LIN {X 0,Y 524.033,Z 442.422,A -85,B 0,C 180,E1 -4780.038,E2 -4780.038} C_VEL
LIN {X 0,Y 524.328,Z 431.907,A -85,B 0,C 180,E1 -4781.009,E2 -4781.009} C_VEL
LIN {X 0,Y 524.611,Z 421.558,A -85,B 0,C 180,E1 -4781.783,E2 -4781.783} C_VEL
LIN {X 0,Y 524.883,Z 410.111,A -85,B 0,C 180,E1 -4782.466,E2 -4782.466} C_VEL
LIN {X 0,Y 525.105,Z 398.418,A -85,B 0,C 180,E1 -4783.001,E2 -4783.001} C_VEL
LIN {X 0,Y 525.367,Z 384.955,A -85,B 0,C 180,E1 -4783.438,E2 -4783.438} C_VEL
LIN {X 0,Y 525.555,Z 371.649,A -85,B 0,C 180,E1 -4783.704,E2 -4783.704} C_VEL
LIN {X 0,Y 525.723,Z 278.906,A -85,B 0,C 180,E1 -4784.981,E2 -4784.981} C_VEL
LIN {X 0,Y 524.283,Z 268.974,A -85,B 0,C 180,E1 -4785.168,E2 -4785.168} C_VEL
LIN {X 0,Y 524.683,Z 247.787,A -85,B 0,C 180,E1 -4788.304,E2 -4788.304} C_VEL
LIN {X 0,Y 525.117,Z 227.261,A -85,B 0,C 180,E1 -4791.386,E2 -4791.386} C_VEL
LIN {X 0,Y 525.445,Z 212.359,A -85,B 0,C 180,E1 -4793.653,E2 -4793.653} C_VEL
LIN {X 0,Y 523.986,Z 204.215,A -85,B 0,C 180,E1 -4794.988,E2 -4794.988} C_VEL
LIN {X 0,Y 523.957,Z 204.223,A -85,B 0,C 180,E1 -4797.995,E2 -4797.995} C_VEL
LIN {X 0,Y 523.928,Z 204.217,A -85,B 0,C 180,E1 -4800.851,E2 -4800.851} C_VEL
LIN {X 0,Y 523.944,Z 204.22,A -85,B 0,C 180,E1 -4803.731,E2 -4803.731} C_VEL
LIN {X 0,Y 523.901,Z 204.224,A -85,B 0,C 180,E1 -4806.4,E2 -4806.4} C_VEL
LIN {X 0,Y 523.899,Z 204.221,A -85,B 0,C 180,E1 -4809.081,E2 -4809.081} C_VEL
LIN {X 0,Y 523.929,Z 204.223,A -85,B 0,C 180,E1 -4812.115,E2 -4812.115} C_VEL
LIN {X 0,Y 523.925,Z 204.219,A -85,B 0,C 180,E1 -4815.305,E2 -4815.305} C_VEL
LIN {X 0,Y 523.949,Z 204.214,A -85,B 0,C 180,E1 -4818.683,E2 -4818.683} C_VEL
LIN {X 0,Y 523.919,Z 204.219,A -85,B 0,C 180,E1 -4821.072,E2 -4821.072} C_VEL
LIN {X 0,Y 523.891,Z 204.229,A -85,B 0,C 180,E1 -4823.824,E2 -4823.824} C_VEL
LIN {X 0,Y 523.902,Z 204.22,A -85,B 0,C 180,E1 -4826.632,E2 -4826.632} C_VEL
LIN {X 0,Y 523.92,Z 204.223,A -85,B 0,C 180,E1 -4829.353,E2 -4829.353} C_VEL
LIN {X 0,Y 523.936,Z 204.217,A -85,B 0,C 180,E1 -4832.277,E2 -4832.277} C_VEL
LIN {X 0,Y 523.908,Z 204.22,A -85,B 0,C 180,E1 -4834.579,E2 -4834.579} C_VEL
LIN {X 0,Y 523.911,Z 204.223,A -85,B 0,C 180,E1 -4837.106,E2 -4837.106} C_VEL
LIN {X 0,Y 523.928,Z 204.22,A -85,B 0,C 180,E1 -4839.863,E2 -4839.863} C_VEL
LIN {X 0,Y 523.945,Z 204.217,A -85,B 0,C 180,E1 -4842.836,E2 -4842.836} C_VEL
LIN {X 0,Y 523.95,Z 204.222,A -85,B 0,C 180,E1 -4845.235,E2 -4845.235} C_VEL
LIN {X 0,Y 523.963,Z 204.213,A -85,B 0,C 180,E1 -4848.393,E2 -4848.393} C_VEL
LIN {X 0,Y 523.954,Z 204.219,A -85,B 0,C 180,E1 -4851.515,E2 -4851.515} C_VEL
LIN {X 0,Y 523.997,Z 204.21,A -85,B 0,C 180,E1 -4853.84,E2 -4853.84} C_VEL
LIN {X 0,Y 524.024,Z 204.211,A -85,B 0,C 180,E1 -4856.925,E2 -4856.925} C_VEL
LIN {X 0,Y 524.051,Z 204.202,A -85,B 0,C 180,E1 -4860,E2 -4860} C_VEL
LIN {X 0,Y 524.022,Z 204.214,A -85,B 0,C 180,E1 -4863.075,E2 -4863.075} C_VEL
LIN {X 0,Y 523.98,Z 204.211,A -85,B 0,C 180,E1 -4866.16,E2 -4866.16} C_VEL
LIN {X 0,Y 523.95,Z 204.218,A -85,B 0,C 180,E1 -4869.262,E2 -4869.262} C_VEL
LIN {X 0,Y 523.968,Z 204.212,A -85,B 0,C 180,E1 -4871.752,E2 -4871.752} C_VEL
LIN {X 0,Y 523.936,Z 204.222,A -85,B 0,C 180,E1 -4875.053,E2 -4875.053} C_VEL
LIN {X 0,Y 523.917,Z 204.219,A -85,B 0,C 180,E1 -4877.97,E2 -4877.97} C_VEL
LIN {X 0,Y 523.92,Z 204.222,A -85,B 0,C 180,E1 -4880.412,E2 -4880.412} C_VEL
LIN {X 0,Y 523.892,Z 204.227,A -85,B 0,C 180,E1 -4882.894,E2 -4882.894} C_VEL
LIN {X 0,Y 523.936,Z 204.217,A -85,B 0,C 180,E1 -4886.022,E2 -4886.022} C_VEL
LIN {X 0,Y 523.895,Z 204.226,A -85,B 0,C 180,E1 -4888.877,E2 -4888.877} C_VEL
LIN {X 0,Y 523.885,Z 204.222,A -85,B 0,C 180,E1 -4891.546,E2 -4891.546} C_VEL
LIN {X 0,Y 523.9,Z 204.227,A -85,B 0,C 180,E1 -4894.292,E2 -4894.292} C_VEL
LIN {X 0,Y 523.871,Z 204.225,A -85,B 0,C 180,E1 -4897.135,E2 -4897.135} C_VEL
LIN {X 0,Y 523.899,Z 204.226,A -85,B 0,C 180,E1 -4900.133,E2 -4900.133} C_VEL
LIN {X 0,Y 523.901,Z 204.228,A -85,B 0,C 180,E1 -4902.462,E2 -4902.462} C_VEL
LIN {X 0,Y 523.91,Z 204.219,A -85,B 0,C 180,E1 -4905.314,E2 -4905.314} C_VEL
LIN {X 0,Y 523.884,Z 204.223,A -85,B 0,C 180,E1 -4906.944,E2 -4906.944} C_VEL
LIN {X 0,Y 523.222,Z 204.306,A -85,B 0,C 180,E1 -4907.585,E2 -4907.585} C_VEL
LIN {X 0,Y 520.38,Z 204.669,A -85,B 0,C 180,E1 -4908.627,E2 -4908.627} C_VEL
LIN {X 0,Y 517.974,Z 204.973,A -85,B 0,C 180,E1 -4909.466,E2 -4909.466} C_VEL
LIN {X 0,Y 516.938,Z 205.098,A -85,B 0,C 180,E1 -4910.114,E2 -4910.114} C_VEL
LIN {X 0,Y 516.852,Z 205.106,A -85,B 0,C 180,E1 -4910.334,E2 -4910.334} C_VEL
LIN {X 0,Y 516.859,Z 205.098,A -85,B 0,C 180,E1 -4913.345,E2 -4913.345} C_VEL
LIN {X 0,Y 516.888,Z 205.103,A -85,B 0,C 180,E1 -4916.124,E2 -4916.124} C_VEL
LIN {X 0,Y 516.871,Z 205.096,A -85,B 0,C 180,E1 -4918.939,E2 -4918.939} C_VEL
LIN {X 0,Y 516.897,Z 205.096,A -85,B 0,C 180,E1 -4921.588,E2 -4921.588} C_VEL
LIN {X 0,Y 516.914,Z 205.096,A -85,B 0,C 180,E1 -4924.214,E2 -4924.214} C_VEL
LIN {X 0,Y 516.846,Z 205.099,A -85,B 0,C 180,E1 -4926.779,E2 -4926.779} C_VEL
LIN {X 0,Y 516.926,Z 205.096,A -85,B 0,C 180,E1 -4929.735,E2 -4929.735} C_VEL
LIN {X 0,Y 516.884,Z 205.095,A -85,B 0,C 180,E1 -4932.598,E2 -4932.598} C_VEL
LIN {X 0,Y 516.928,Z 205.09,A -85,B 0,C 180,E1 -4935.032,E2 -4935.032} C_VEL
LIN {X 0,Y 516.961,Z 205.087,A -85,B 0,C 180,E1 -4938.236,E2 -4938.236} C_VEL
LIN {X 0,Y 516.959,Z 205.09,A -85,B 0,C 180,E1 -4941.402,E2 -4941.402} C_VEL
LIN {X 0,Y 517.019,Z 205.081,A -85,B 0,C 180,E1 -4944.542,E2 -4944.542} C_VEL
LIN {X 0,Y 516.866,Z 205.164,A -85,B 0,C 180,E1 -4946.006,E2 -4946.006} C_VEL
LIN {X 0,Y 517.422,Z 209.6,A -85,B 0,C 180,E1 -4946.887,E2 -4946.887} C_VEL
LIN {X 0,Y 517.24,Z 224.307,A -85,B 0,C 180,E1 -4949.697,E2 -4949.697} C_VEL
LIN {X 0,Y 519.169,Z 234.742,A -85,B 0,C 180,E1 -4949.904,E2 -4949.904} C_VEL
LIN {X 0,Y 518.648,Z 331.01,A -85,B 0,C 180,E1 -4951.263,E2 -4951.263} C_VEL
LIN {X 0,Y 518.467,Z 343.297,A -85,B 0,C 180,E1 -4951.579,E2 -4951.579} C_VEL
LIN {X 0,Y 518.269,Z 356.555,A -85,B 0,C 180,E1 -4952.09,E2 -4952.09} C_VEL
LIN {X 0,Y 517.968,Z 368.557,A -85,B 0,C 180,E1 -4952.723,E2 -4952.723} C_VEL
LIN {X 0,Y 517.629,Z 379.969,A -85,B 0,C 180,E1 -4953.504,E2 -4953.504} C_VEL
LIN {X 0,Y 517.351,Z 390.246,A -85,B 0,C 180,E1 -4954.383,E2 -4954.383} C_VEL
LIN {X 0,Y 517.064,Z 398.689,A -85,B 0,C 180,E1 -4955.265,E2 -4955.265} C_VEL
LIN {X 0,Y 516.856,Z 406.477,A -85,B 0,C 180,E1 -4956.246,E2 -4956.246} C_VEL
LIN {X 0,Y 516.683,Z 414.099,A -85,B 0,C 180,E1 -4957.425,E2 -4957.425} C_VEL
LIN {X 0,Y 516.521,Z 420.242,A -85,B 0,C 180,E1 -4958.608,E2 -4958.608} C_VEL
LIN {X 0,Y 516.42,Z 425.127,A -85,B 0,C 180,E1 -4959.795,E2 -4959.795} C_VEL
LIN {X 0,Y 516.338,Z 428.896,A -85,B 0,C 180,E1 -4960.986,E2 -4960.986} C_VEL
LIN {X 0,Y 516.291,Z 430.844,A -85,B 0,C 180,E1 -4961.782,E2 -4961.782} C_VEL
LIN {X 0,Y 516.23,Z 432.359,A -85,B 0,C 180,E1 -4962.582,E2 -4962.582} C_VEL
LIN {X 0,Y 516.205,Z 433.411,A -85,B 0,C 180,E1 -4963.383,E2 -4963.383} C_VEL
LIN {X 0,Y 516.249,Z 434.294,A -85,B 0,C 180,E1 -4964.859,E2 -4964.859} C_VEL
LIN {X 0,Y 516.174,Z 434.133,A -85,B 0,C 180,E1 -4965.802,E2 -4965.802} C_VEL
LIN {X 0,Y 516.195,Z 433.514,A -85,B 0,C 180,E1 -4966.613,E2 -4966.613} C_VEL
LIN {X 0,Y 516.247,Z 432.135,A -85,B 0,C 180,E1 -4967.645,E2 -4967.645} C_VEL
LIN {X 0,Y 516.303,Z 429.017,A -85,B 0,C 180,E1 -4969.068,E2 -4969.068} C_VEL
LIN {X 0,Y 516.402,Z 424.901,A -85,B 0,C 180,E1 -4970.367,E2 -4970.367} C_VEL
LIN {X 0,Y 516.481,Z 419.948,A -85,B 0,C 180,E1 -4971.555,E2 -4971.555} C_VEL
LIN {X 0,Y 516.685,Z 413.32,A -85,B 0,C 180,E1 -4972.808,E2 -4972.808} C_VEL
LIN {X 0,Y 516.912,Z 404.823,A -85,B 0,C 180,E1 -4974.071,E2 -4974.071} C_VEL
LIN {X 0,Y 517.164,Z 396.005,A -85,B 0,C 180,E1 -4975.129,E2 -4975.129} C_VEL
LIN {X 0,Y 517.466,Z 386.153,A -85,B 0,C 180,E1 -4976.087,E2 -4976.087} C_VEL
LIN {X 0,Y 517.771,Z 375.246,A -85,B 0,C 180,E1 -4976.936,E2 -4976.936} C_VEL
LIN {X 0,Y 518.116,Z 363.348,A -85,B 0,C 180,E1 -4977.668,E2 -4977.668} C_VEL
LIN {X 0,Y 518.317,Z 352.206,A -85,B 0,C 180,E1 -4978.195,E2 -4978.195} C_VEL
LIN {X 0,Y 518.52,Z 339.67,A -85,B 0,C 180,E1 -4978.622,E2 -4978.622} C_VEL
LIN {X 0,Y 518.636,Z 326.636,A -85,B 0,C 180,E1 -4978.905,E2 -4978.905} C_VEL
LIN {X 0,Y 519.051,Z 233.834,A -85,B 0,C 180,E1 -4980.204,E2 -4980.204} C_VEL
LIN {X 0,Y 517.237,Z 224.156,A -85,B 0,C 180,E1 -4980.397,E2 -4980.397} C_VEL
LIN {X 0,Y 517.378,Z 209.592,A -85,B 0,C 180,E1 -4983.143,E2 -4983.143} C_VEL
LIN {X 0,Y 516.965,Z 205.092,A -85,B 0,C 180,E1 -4984.019,E2 -4984.019} C_VEL
LIN {X 0,Y 516.873,Z 205.103,A -85,B 0,C 180,E1 -4986.744,E2 -4986.744} C_VEL
LIN {X 0,Y 516.891,Z 205.098,A -85,B 0,C 180,E1 -4989.718,E2 -4989.718} C_VEL
LIN {X 0,Y 516.894,Z 205.099,A -85,B 0,C 180,E1 -4992.759,E2 -4992.759} C_VEL
LIN {X 0,Y 516.907,Z 205.094,A -85,B 0,C 180,E1 -4995.009,E2 -4995.009} C_VEL
LIN {X 0,Y 516.905,Z 205.099,A -85,B 0,C 180,E1 -4998.396,E2 -4998.396} C_VEL
LIN {X 0,Y 516.866,Z 205.098,A -85,B 0,C 180,E1 -5001.283,E2 -5001.283} C_VEL
LIN {X 0,Y 516.869,Z 205.102,A -85,B 0,C 180,E1 -5004.22,E2 -5004.22} C_VEL
LIN {X 0,Y 516.875,Z 205.096,A -85,B 0,C 180,E1 -5007.052,E2 -5007.052} C_VEL
LIN {X 0,Y 516.877,Z 205.102,A -85,B 0,C 180,E1 -5009.796,E2 -5009.796} C_VEL
LIN {X 0,Y 516.904,Z 205.093,A -85,B 0,C 180,E1 -5012.466,E2 -5012.466} C_VEL
LIN {X 0,Y 516.893,Z 205.092,A -85,B 0,C 180,E1 -5015.071,E2 -5015.071} C_VEL
LIN {X 0,Y 516.884,Z 205.102,A -85,B 0,C 180,E1 -5017.622,E2 -5017.622} C_VEL
LIN {X 0,Y 516.902,Z 205.095,A -85,B 0,C 180,E1 -5020.129,E2 -5020.129} C_VEL
LIN {X 0,Y 516.912,Z 205.089,A -85,B 0,C 180,E1 -5022.596,E2 -5022.596} C_VEL
LIN {X 0,Y 516.918,Z 205.093,A -85,B 0,C 180,E1 -5025.03,E2 -5025.03} C_VEL
LIN {X 0,Y 516.933,Z 205.089,A -85,B 0,C 180,E1 -5028.233,E2 -5028.233} C_VEL
LIN {X 0,Y 516.94,Z 205.093,A -85,B 0,C 180,E1 -5031.399,E2 -5031.399} C_VEL
LIN {X 0,Y 516.985,Z 205.085,A -85,B 0,C 180,E1 -5033.757,E2 -5033.757} C_VEL
LIN {X 0,Y 516.984,Z 205.082,A -85,B 0,C 180,E1 -5036.883,E2 -5036.883} C_VEL
LIN {X 0,Y 517.044,Z 205.073,A -85,B 0,C 180,E1 -5040,E2 -5040} C_VEL
LIN {X 0,Y 516.982,Z 205.088,A -85,B 0,C 180,E1 -5043.117,E2 -5043.117} C_VEL
LIN {X 0,Y 516.967,Z 205.081,A -85,B 0,C 180,E1 -5046.244,E2 -5046.244} C_VEL
LIN {X 0,Y 516.921,Z 205.09,A -85,B 0,C 180,E1 -5049.39,E2 -5049.39} C_VEL
LIN {X 0,Y 516.952,Z 205.085,A -85,B 0,C 180,E1 -5051.825,E2 -5051.825} C_VEL
LIN {X 0,Y 516.912,Z 205.096,A -85,B 0,C 180,E1 -5055.147,E2 -5055.147} C_VEL
LIN {X 0,Y 516.885,Z 205.095,A -85,B 0,C 180,E1 -5058.224,E2 -5058.224} C_VEL
LIN {X 0,Y 516.883,Z 205.101,A -85,B 0,C 180,E1 -5060.703,E2 -5060.703} C_VEL
LIN {X 0,Y 516.855,Z 205.098,A -85,B 0,C 180,E1 -5064.075,E2 -5064.075} C_VEL
LIN {X 0,Y 516.866,Z 205.104,A -85,B 0,C 180,E1 -5066.661,E2 -5066.661} C_VEL
LIN {X 0,Y 516.883,Z 205.095,A -85,B 0,C 180,E1 -5069.525,E2 -5069.525} C_VEL
LIN {X 0,Y 516.871,Z 205.105,A -85,B 0,C 180,E1 -5072.545,E2 -5072.545} C_VEL
LIN {X 0,Y 516.841,Z 205.101,A -85,B 0,C 180,E1 -5075.331,E2 -5075.331} C_VEL
LIN {X 0,Y 516.857,Z 205.1,A -85,B 0,C 180,E1 -5077.944,E2 -5077.944} C_VEL
LIN {X 0,Y 516.867,Z 205.097,A -85,B 0,C 180,E1 -5080.744,E2 -5080.744} C_VEL
LIN {X 0,Y 516.867,Z 205.099,A -85,B 0,C 180,E1 -5082.833,E2 -5082.833} C_VEL
LIN {X 0,Y 516.882,Z 205.096,A -85,B 0,C 180,E1 -5085.009,E2 -5085.009} C_VEL
LIN {X 0,Y 516.89,Z 205.1,A -85,B 0,C 180,E1 -5088.402,E2 -5088.402} C_VEL
LIN {X 0,Y 516.867,Z 205.098,A -85,B 0,C 180,E1 -5091.285,E2 -5091.285} C_VEL
LIN {X 0,Y 516.868,Z 205.105,A -85,B 0,C 180,E1 -5094.222,E2 -5094.222} C_VEL
LIN {X 0,Y 516.889,Z 205.096,A -85,B 0,C 180,E1 -5097.054,E2 -5097.054} C_VEL
LIN {X 0,Y 516.887,Z 205.101,A -85,B 0,C 180,E1 -5099.798,E2 -5099.798} C_VEL
LIN {X 0,Y 516.895,Z 205.099,A -85,B 0,C 180,E1 -5102.467,E2 -5102.467} C_VEL
LIN {X 0,Y 516.93,Z 205.133,A -85,B 0,C 180,E1 -5104.913,E2 -5104.913} C_VEL
LIN {X 0,Y 518.493,Z 214.374,A -85,B 0,C 180,E1 -5106.431,E2 -5106.431} C_VEL
LIN {X 0,Y 517.974,Z 234.682,A -85,B 0,C 180,E1 -5109.539,E2 -5109.539} C_VEL
LIN {X 0,Y 517.563,Z 253.888,A -85,B 0,C 180,E1 -5112.437,E2 -5112.437} C_VEL
LIN {X 0,Y 517.227,Z 268.524,A -85,B 0,C 180,E1 -5114.62,E2 -5114.62} C_VEL
LIN {X 0,Y 519.024,Z 282.03,A -85,B 0,C 180,E1 -5114.87,E2 -5114.87} C_VEL
LIN {X 0,Y 518.593,Z 376.948,A -85,B 0,C 180,E1 -5116.206,E2 -5116.206} C_VEL
LIN {X 0,Y 518.326,Z 390.326,A -85,B 0,C 180,E1 -5116.548,E2 -5116.548} C_VEL
LIN {X 0,Y 518.033,Z 402.555,A -85,B 0,C 180,E1 -5117.015,E2 -5117.015} C_VEL
LIN {X 0,Y 517.801,Z 414.873,A -85,B 0,C 180,E1 -5117.655,E2 -5117.655} C_VEL
LIN {X 0,Y 517.468,Z 426.547,A -85,B 0,C 180,E1 -5118.444,E2 -5118.444} C_VEL
LIN {X 0,Y 517.209,Z 437.038,A -85,B 0,C 180,E1 -5119.33,E2 -5119.33} C_VEL
LIN {X 0,Y 516.917,Z 445.615,A -85,B 0,C 180,E1 -5120.215,E2 -5120.215} C_VEL
LIN {X 0,Y 516.703,Z 453.533,A -85,B 0,C 180,E1 -5121.198,E2 -5121.198} C_VEL
LIN {X 0,Y 516.521,Z 461.27,A -85,B 0,C 180,E1 -5122.376,E2 -5122.376} C_VEL
LIN {X 0,Y 516.389,Z 468.402,A -85,B 0,C 180,E1 -5123.749,E2 -5123.749} C_VEL
LIN {X 0,Y 516.312,Z 473.149,A -85,B 0,C 180,E1 -5124.923,E2 -5124.923} C_VEL
LIN {X 0,Y 516.352,Z 476.781,A -85,B 0,C 180,E1 -5126.097,E2 -5126.097} C_VEL
LIN {X 0,Y 516.283,Z 478.651,A -85,B 0,C 180,E1 -5126.878,E2 -5126.878} C_VEL
LIN {X 0,Y 516.262,Z 480.055,A -85,B 0,C 180,E1 -5127.658,E2 -5127.658} C_VEL
LIN {X 0,Y 516.167,Z 481.667,A -85,B 0,C 180,E1 -5129.219,E2 -5129.219} C_VEL
LIN {X 0,Y 516.167,Z 481.887,A -85,B 0,C 180,E1 -5129.999,E2 -5129.999} C_VEL
LIN {X 0,Y 516.192,Z 481.066,A -85,B 0,C 180,E1 -5131.559,E2 -5131.559} C_VEL
LIN {X 0,Y 516.261,Z 480.072,A -85,B 0,C 180,E1 -5132.339,E2 -5132.339} C_VEL
LIN {X 0,Y 516.282,Z 478.673,A -85,B 0,C 180,E1 -5133.12,E2 -5133.12} C_VEL
LIN {X 0,Y 516.311,Z 475.73,A -85,B 0,C 180,E1 -5134.292,E2 -5134.292} C_VEL
LIN {X 0,Y 516.368,Z 471.744,A -85,B 0,C 180,E1 -5135.465,E2 -5135.465} C_VEL
LIN {X 0,Y 516.387,Z 466.554,A -85,B 0,C 180,E1 -5136.653,E2 -5136.653} C_VEL
LIN {X 0,Y 516.543,Z 460.155,A -85,B 0,C 180,E1 -5137.818,E2 -5137.818} C_VEL
LIN {X 0,Y 516.752,Z 452.102,A -85,B 0,C 180,E1 -5138.996,E2 -5138.996} C_VEL
LIN {X 0,Y 516.948,Z 443.896,A -85,B 0,C 180,E1 -5139.98,E2 -5139.98} C_VEL
LIN {X 0,Y 517.262,Z 433.895,A -85,B 0,C 180,E1 -5140.963,E2 -5140.963} C_VEL
LIN {X 0,Y 517.524,Z 424.03,A -85,B 0,C 180,E1 -5141.751,E2 -5141.751} C_VEL
LIN {X 0,Y 517.84,Z 412.87,A -85,B 0,C 180,E1 -5142.465,E2 -5142.465} C_VEL
LIN {X 0,Y 518.16,Z 400.426,A -85,B 0,C 180,E1 -5143.079,E2 -5143.079} C_VEL
LIN {X 0,Y 518.419,Z 388.196,A -85,B 0,C 180,E1 -5143.521,E2 -5143.521} C_VEL
LIN {X 0,Y 518.602,Z 375.803,A -85,B 0,C 180,E1 -5143.816,E2 -5143.816} C_VEL
LIN {X 0,Y 519.017,Z 281.094,A -85,B 0,C 180,E1 -5145.145,E2 -5145.145} C_VEL
LIN {X 0,Y 517.229,Z 268.643,A -85,B 0,C 180,E1 -5145.381,E2 -5145.381} C_VEL
LIN {X 0,Y 517.637,Z 249.904,A -85,B 0,C 180,E1 -5148.193,E2 -5148.193} C_VEL
LIN {X 0,Y 518.13,Z 229.636,A -85,B 0,C 180,E1 -5151.271,E2 -5151.271} C_VEL
LIN {X 0,Y 518.562,Z 214.731,A -85,B 0,C 180,E1 -5153.562,E2 -5153.562} C_VEL
LIN {X 0,Y 516.939,Z 205.093,A -85,B 0,C 180,E1 -5155.151,E2 -5155.151} C_VEL
LIN {X 0,Y 516.914,Z 205.099,A -85,B 0,C 180,E1 -5157.902,E2 -5157.902} C_VEL
LIN {X 0,Y 516.877,Z 205.103,A -85,B 0,C 180,E1 -5160.2,E2 -5160.2} C_VEL
LIN {X 0,Y 516.879,Z 205.095,A -85,B 0,C 180,E1 -5162.943,E2 -5162.943} C_VEL
LIN {X 0,Y 516.87,Z 205.102,A -85,B 0,C 180,E1 -5165.775,E2 -5165.775} C_VEL
LIN {X 0,Y 516.859,Z 205.098,A -85,B 0,C 180,E1 -5168.712,E2 -5168.712} C_VEL
LIN {X 0,Y 516.888,Z 205.101,A -85,B 0,C 180,E1 -5171.771,E2 -5171.771} C_VEL
LIN {X 0,Y 516.893,Z 205.094,A -85,B 0,C 180,E1 -5175.006,E2 -5175.006} C_VEL
LIN {X 0,Y 516.897,Z 205.094,A -85,B 0,C 180,E1 -5178.393,E2 -5178.393} C_VEL
LIN {X 0,Y 516.871,Z 205.099,A -85,B 0,C 180,E1 -5181.283,E2 -5181.283} C_VEL
LIN {X 0,Y 516.853,Z 205.1,A -85,B 0,C 180,E1 -5184.218,E2 -5184.218} C_VEL
LIN {X 0,Y 516.857,Z 205.099,A -85,B 0,C 180,E1 -5187.05,E2 -5187.05} C_VEL
LIN {X 0,Y 516.859,Z 205.104,A -85,B 0,C 180,E1 -5189.794,E2 -5189.794} C_VEL
LIN {X 0,Y 516.885,Z 205.094,A -85,B 0,C 180,E1 -5192.465,E2 -5192.465} C_VEL
LIN {X 0,Y 516.876,Z 205.099,A -85,B 0,C 180,E1 -5195.07,E2 -5195.07} C_VEL
LIN {X 0,Y 516.863,Z 205.104,A -85,B 0,C 180,E1 -5197.621,E2 -5197.621} C_VEL
LIN {X 0,Y 516.881,Z 205.096,A -85,B 0,C 180,E1 -5200.128,E2 -5200.128} C_VEL
LIN {X 0,Y 516.891,Z 205.094,A -85,B 0,C 180,E1 -5202.595,E2 -5202.595} C_VEL
LIN {X 0,Y 516.856,Z 205.1,A -85,B 0,C 180,E1 -5205.832,E2 -5205.832} C_VEL
LIN {X 0,Y 516.949,Z 205.086,A -85,B 0,C 180,E1 -5208.233,E2 -5208.233} C_VEL
LIN {X 0,Y 516.918,Z 205.097,A -85,B 0,C 180,E1 -5211.399,E2 -5211.399} C_VEL
LIN {X 0,Y 516.965,Z 205.086,A -85,B 0,C 180,E1 -5213.756,E2 -5213.756} C_VEL
LIN {X 0,Y 516.964,Z 205.09,A -85,B 0,C 180,E1 -5216.883,E2 -5216.883} C_VEL
LIN {X 0,Y 517.022,Z 205.077,A -85,B 0,C 180,E1 -5220,E2 -5220} C_VEL
LIN {X 0,Y 516.963,Z 205.092,A -85,B 0,C 180,E1 -5223.117,E2 -5223.117} C_VEL
LIN {X 0,Y 516.945,Z 205.088,A -85,B 0,C 180,E1 -5226.244,E2 -5226.244} C_VEL
LIN {X 0,Y 516.905,Z 205.094,A -85,B 0,C 180,E1 -5229.39,E2 -5229.39} C_VEL
LIN {X 0,Y 516.927,Z 205.089,A -85,B 0,C 180,E1 -5231.825,E2 -5231.825} C_VEL
LIN {X 0,Y 516.888,Z 205.098,A -85,B 0,C 180,E1 -5235.147,E2 -5235.147} C_VEL
LIN {X 0,Y 516.876,Z 205.097,A -85,B 0,C 180,E1 -5238.224,E2 -5238.224} C_VEL
LIN {X 0,Y 516.863,Z 205.106,A -85,B 0,C 180,E1 -5240.703,E2 -5240.703} C_VEL
LIN {X 0,Y 516.84,Z 205.102,A -85,B 0,C 180,E1 -5243.225,E2 -5243.225} C_VEL
LIN {X 0,Y 516.895,Z 205.096,A -85,B 0,C 180,E1 -5246.199,E2 -5246.199} C_VEL
LIN {X 0,Y 516.876,Z 205.096,A -85,B 0,C 180,E1 -5249.307,E2 -5249.307} C_VEL
LIN {X 0,Y 516.855,Z 205.107,A -85,B 0,C 180,E1 -5252.547,E2 -5252.547} C_VEL
LIN {X 0,Y 516.84,Z 205.1,A -85,B 0,C 180,E1 -5255.335,E2 -5255.335} C_VEL
LIN {X 0,Y 516.84,Z 205.102,A -85,B 0,C 180,E1 -5257.946,E2 -5257.946} C_VEL
LIN {X 0,Y 516.849,Z 205.103,A -85,B 0,C 180,E1 -5260.745,E2 -5260.745} C_VEL
LIN {X 0,Y 516.848,Z 205.101,A -85,B 0,C 180,E1 -5262.835,E2 -5262.835} C_VEL
LIN {X 0,Y 516.861,Z 205.098,A -85,B 0,C 180,E1 -5265.01,E2 -5265.01} C_VEL
LIN {X 0,Y 516.887,Z 205.101,A -85,B 0,C 180,E1 -5268.402,E2 -5268.402} C_VEL
LIN {X 0,Y 516.852,Z 205.106,A -85,B 0,C 180,E1 -5270.334,E2 -5270.334} C_VEL
LIN {X 0,Y 516.183,Z 205.184,A -85,B 0,C 180,E1 -5270.984,E2 -5270.984} C_VEL
LIN {X 0,Y 513.338,Z 205.543,A -85,B 0,C 180,E1 -5272.04,E2 -5272.04} C_VEL
LIN {X 0,Y 510.931,Z 205.841,A -85,B 0,C 180,E1 -5272.89,E2 -5272.89} C_VEL
LIN {X 0,Y 509.892,Z 205.968,A -85,B 0,C 180,E1 -5273.547,E2 -5273.547} C_VEL
LIN {X 0,Y 509.804,Z 205.978,A -85,B 0,C 180,E1 -5273.769,E2 -5273.769} C_VEL
LIN {X 0,Y 509.838,Z 205.975,A -85,B 0,C 180,E1 -5276.543,E2 -5276.543} C_VEL
LIN {X 0,Y 509.826,Z 205.974,A -85,B 0,C 180,E1 -5279.338,E2 -5279.338} C_VEL
LIN {X 0,Y 509.872,Z 205.977,A -85,B 0,C 180,E1 -5282.058,E2 -5282.058} C_VEL
LIN {X 0,Y 509.825,Z 205.975,A -85,B 0,C 180,E1 -5284.705,E2 -5284.705} C_VEL
LIN {X 0,Y 509.813,Z 205.978,A -85,B 0,C 180,E1 -5287.461,E2 -5287.461} C_VEL
LIN {X 0,Y 509.903,Z 205.973,A -85,B 0,C 180,E1 -5289.848,E2 -5289.848} C_VEL
LIN {X 0,Y 509.853,Z 205.972,A -85,B 0,C 180,E1 -5293.177,E2 -5293.177} C_VEL
LIN {X 0,Y 509.847,Z 205.978,A -85,B 0,C 180,E1 -5295.636,E2 -5295.636} C_VEL
LIN {X 0,Y 509.906,Z 205.964,A -85,B 0,C 180,E1 -5298.877,E2 -5298.877} C_VEL
LIN {X 0,Y 509.915,Z 205.968,A -85,B 0,C 180,E1 -5302.08,E2 -5302.08} C_VEL
LIN {X 0,Y 509.97,Z 205.96,A -85,B 0,C 180,E1 -5304.466,E2 -5304.466} C_VEL
LIN {X 0,Y 509.86,Z 206.116,A -85,B 0,C 180,E1 -5305.901,E2 -5305.901} C_VEL
LIN {X 0,Y 510.435,Z 210.814,A -85,B 0,C 180,E1 -5306.845,E2 -5306.845} C_VEL
LIN {X 0,Y 510.286,Z 224.635,A -85,B 0,C 180,E1 -5309.484,E2 -5309.484} C_VEL
LIN {X 0,Y 512.352,Z 235.662,A -85,B 0,C 180,E1 -5309.707,E2 -5309.707} C_VEL
LIN {X 0,Y 511.749,Z 331.728,A -85,B 0,C 180,E1 -5311.083,E2 -5311.083} C_VEL
LIN {X 0,Y 511.572,Z 344.607,A -85,B 0,C 180,E1 -5311.428,E2 -5311.428} C_VEL
LIN {X 0,Y 511.351,Z 357.068,A -85,B 0,C 180,E1 -5311.921,E2 -5311.921} C_VEL
LIN {X 0,Y 511.044,Z 369.007,A -85,B 0,C 180,E1 -5312.563,E2 -5312.563} C_VEL
LIN {X 0,Y 510.663,Z 380.405,A -85,B 0,C 180,E1 -5313.354,E2 -5313.354} C_VEL
LIN {X 0,Y 510.372,Z 390.661,A -85,B 0,C 180,E1 -5314.246,E2 -5314.246} C_VEL
LIN {X 0,Y 510.064,Z 399.09,A -85,B 0,C 180,E1 -5315.139,E2 -5315.139} C_VEL
LIN {X 0,Y 509.849,Z 406.861,A -85,B 0,C 180,E1 -5316.133,E2 -5316.133} C_VEL
LIN {X 0,Y 509.648,Z 414.471,A -85,B 0,C 180,E1 -5317.329,E2 -5317.329} C_VEL
LIN {X 0,Y 509.439,Z 421.512,A -85,B 0,C 180,E1 -5318.729,E2 -5318.729} C_VEL
LIN {X 0,Y 509.322,Z 426.202,A -85,B 0,C 180,E1 -5319.933,E2 -5319.933} C_VEL
LIN {X 0,Y 509.274,Z 429.781,A -85,B 0,C 180,E1 -5321.14,E2 -5321.14} C_VEL
LIN {X 0,Y 509.208,Z 431.611,A -85,B 0,C 180,E1 -5321.948,E2 -5321.948} C_VEL
LIN {X 0,Y 509.142,Z 432.982,A -85,B 0,C 180,E1 -5322.76,E2 -5322.76} C_VEL
LIN {X 0,Y 509.112,Z 433.951,A -85,B 0,C 180,E1 -5323.573,E2 -5323.573} C_VEL
LIN {X 0,Y 509.15,Z 434.637,A -85,B 0,C 180,E1 -5324.932,E2 -5324.932} C_VEL
LIN {X 0,Y 509.079,Z 434.331,A -85,B 0,C 180,E1 -5326.028,E2 -5326.028} C_VEL
LIN {X 0,Y 509.126,Z 433.626,A -85,B 0,C 180,E1 -5326.851,E2 -5326.851} C_VEL
LIN {X 0,Y 509.174,Z 432.335,A -85,B 0,C 180,E1 -5327.752,E2 -5327.752} C_VEL
LIN {X 0,Y 509.218,Z 429.873,A -85,B 0,C 180,E1 -5328.925,E2 -5328.925} C_VEL
LIN {X 0,Y 509.311,Z 425.988,A -85,B 0,C 180,E1 -5330.227,E2 -5330.227} C_VEL
LIN {X 0,Y 509.407,Z 421.183,A -85,B 0,C 180,E1 -5331.444,E2 -5331.444} C_VEL
LIN {X 0,Y 509.626,Z 414.787,A -85,B 0,C 180,E1 -5332.713,E2 -5332.713} C_VEL
LIN {X 0,Y 509.82,Z 408.137,A -85,B 0,C 180,E1 -5333.779,E2 -5333.779} C_VEL
LIN {X 0,Y 510.09,Z 399.797,A -85,B 0,C 180,E1 -5334.875,E2 -5334.875} C_VEL
LIN {X 0,Y 510.418,Z 389.897,A -85,B 0,C 180,E1 -5335.922,E2 -5335.922} C_VEL
LIN {X 0,Y 510.752,Z 378.876,A -85,B 0,C 180,E1 -5336.86,E2 -5336.86} C_VEL
LIN {X 0,Y 511.078,Z 368.875,A -85,B 0,C 180,E1 -5337.54,E2 -5337.54} C_VEL
LIN {X 0,Y 511.339,Z 356.877,A -85,B 0,C 180,E1 -5338.182,E2 -5338.182} C_VEL
LIN {X 0,Y 511.556,Z 344.005,A -85,B 0,C 180,E1 -5338.686,E2 -5338.686} C_VEL
LIN {X 0,Y 511.7,Z 331.679,A -85,B 0,C 180,E1 -5339.011,E2 -5339.011} C_VEL
LIN {X 0,Y 512.211,Z 234.636,A -85,B 0,C 180,E1 -5340.405,E2 -5340.405} C_VEL
LIN {X 0,Y 510.262,Z 224.324,A -85,B 0,C 180,E1 -5340.636,E2 -5340.636} C_VEL
LIN {X 0,Y 510.414,Z 211.299,A -85,B 0,C 180,E1 -5343.099,E2 -5343.099} C_VEL
LIN {X 0,Y 510.006,Z 206.488,A -85,B 0,C 180,E1 -5344.03,E2 -5344.03} C_VEL
LIN {X 0,Y 509.929,Z 205.969,A -85,B 0,C 180,E1 -5344.215,E2 -5344.215} C_VEL
LIN {X 0,Y 509.809,Z 205.979,A -85,B 0,C 180,E1 -5347.339,E2 -5347.339} C_VEL
LIN {X 0,Y 509.85,Z 205.979,A -85,B 0,C 180,E1 -5350.378,E2 -5350.378} C_VEL
LIN {X 0,Y 509.826,Z 205.977,A -85,B 0,C 180,E1 -5353.063,E2 -5353.063} C_VEL
LIN {X 0,Y 509.814,Z 205.98,A -85,B 0,C 180,E1 -5355.791,E2 -5355.791} C_VEL
LIN {X 0,Y 509.848,Z 205.975,A -85,B 0,C 180,E1 -5358.574,E2 -5358.574} C_VEL
LIN {X 0,Y 509.832,Z 205.979,A -85,B 0,C 180,E1 -5361.785,E2 -5361.785} C_VEL
LIN {X 0,Y 509.824,Z 205.975,A -85,B 0,C 180,E1 -5364.622,E2 -5364.622} C_VEL
LIN {X 0,Y 509.843,Z 205.975,A -85,B 0,C 180,E1 -5367.48,E2 -5367.48} C_VEL
LIN {X 0,Y 509.857,Z 205.973,A -85,B 0,C 180,E1 -5370.268,E2 -5370.268} C_VEL
LIN {X 0,Y 509.861,Z 205.969,A -85,B 0,C 180,E1 -5372.943,E2 -5372.943} C_VEL
LIN {X 0,Y 509.861,Z 205.973,A -85,B 0,C 180,E1 -5375.574,E2 -5375.574} C_VEL
LIN {X 0,Y 509.826,Z 205.974,A -85,B 0,C 180,E1 -5378.149,E2 -5378.149} C_VEL
LIN {X 0,Y 509.837,Z 205.973,A -85,B 0,C 180,E1 -5380.681,E2 -5380.681} C_VEL
LIN {X 0,Y 509.871,Z 205.969,A -85,B 0,C 180,E1 -5383.175,E2 -5383.175} C_VEL
LIN {X 0,Y 509.842,Z 205.979,A -85,B 0,C 180,E1 -5385.634,E2 -5385.634} C_VEL
LIN {X 0,Y 509.886,Z 205.967,A -85,B 0,C 180,E1 -5388.874,E2 -5388.874} C_VEL
LIN {X 0,Y 509.925,Z 205.96,A -85,B 0,C 180,E1 -5392.078,E2 -5392.078} C_VEL
LIN {X 0,Y 509.964,Z 205.956,A -85,B 0,C 180,E1 -5394.464,E2 -5394.464} C_VEL
LIN {X 0,Y 510.019,Z 205.953,A -85,B 0,C 180,E1 -5397.631,E2 -5397.631} C_VEL
LIN {X 0,Y 510.016,Z 205.948,A -85,B 0,C 180,E1 -5400,E2 -5400} C_VEL
LIN {X 0,Y 510.017,Z 205.948,A -85,B 0,C 180,E1 -5402.37,E2 -5402.37} C_VEL
LIN {X 0,Y 509.945,Z 205.958,A -85,B 0,C 180,E1 -5405.536,E2 -5405.536} C_VEL
LIN {X 0,Y 509.887,Z 205.965,A -85,B 0,C 180,E1 -5407.923,E2 -5407.923} C_VEL
LIN {X 0,Y 509.901,Z 205.97,A -85,B 0,C 180,E1 -5411.126,E2 -5411.126} C_VEL
LIN {X 0,Y 509.828,Z 205.973,A -85,B 0,C 180,E1 -5414.367,E2 -5414.367} C_VEL
LIN {X 0,Y 509.841,Z 205.979,A -85,B 0,C 180,E1 -5416.827,E2 -5416.827} C_VEL
LIN {X 0,Y 509.887,Z 205.966,A -85,B 0,C 180,E1 -5420.157,E2 -5420.157} C_VEL
LIN {X 0,Y 509.789,Z 205.977,A -85,B 0,C 180,E1 -5423.566,E2 -5423.566} C_VEL
LIN {X 0,Y 509.846,Z 205.977,A -85,B 0,C 180,E1 -5426.371,E2 -5426.371} C_VEL
LIN {X 0,Y 509.834,Z 205.974,A -85,B 0,C 180,E1 -5429.728,E2 -5429.728} C_VEL
LIN {X 0,Y 509.822,Z 205.98,A -85,B 0,C 180,E1 -5432.771,E2 -5432.771} C_VEL
LIN {X 0,Y 509.801,Z 205.978,A -85,B 0,C 180,E1 -5435.579,E2 -5435.579} C_VEL
LIN {X 0,Y 509.828,Z 205.98,A -85,B 0,C 180,E1 -5438.34,E2 -5438.34} C_VEL
LIN {X 0,Y 509.84,Z 205.968,A -85,B 0,C 180,E1 -5441.427,E2 -5441.427} C_VEL
LIN {X 0,Y 509.825,Z 205.978,A -85,B 0,C 180,E1 -5444.672,E2 -5444.672} C_VEL
LIN {X 0,Y 509.834,Z 205.98,A -85,B 0,C 180,E1 -5448.107,E2 -5448.107} C_VEL
LIN {X 0,Y 509.823,Z 205.978,A -85,B 0,C 180,E1 -5450.648,E2 -5450.648} C_VEL
LIN {X 0,Y 509.819,Z 205.977,A -85,B 0,C 180,E1 -5453.649,E2 -5453.649} C_VEL
LIN {X 0,Y 509.854,Z 205.975,A -85,B 0,C 180,E1 -5456.541,E2 -5456.541} C_VEL
LIN {X 0,Y 509.841,Z 205.976,A -85,B 0,C 180,E1 -5459.336,E2 -5459.336} C_VEL
LIN {X 0,Y 509.845,Z 205.979,A -85,B 0,C 180,E1 -5462.053,E2 -5462.053} C_VEL
LIN {X 0,Y 509.897,Z 206.176,A -85,B 0,C 180,E1 -5464.753,E2 -5464.753} C_VEL
LIN {X 0,Y 511.557,Z 215.459,A -85,B 0,C 180,E1 -5466.307,E2 -5466.307} C_VEL
LIN {X 0,Y 511.021,Z 235.178,A -85,B 0,C 180,E1 -5469.375,E2 -5469.375} C_VEL
LIN {X 0,Y 510.545,Z 254.763,A -85,B 0,C 180,E1 -5472.372,E2 -5472.372} C_VEL
LIN {X 0,Y 510.234,Z 268.187,A -85,B 0,C 180,E1 -5474.405,E2 -5474.405} C_VEL
LIN {X 0,Y 512.184,Z 281.337,A -85,B 0,C 180,E1 -5474.659,E2 -5474.659} C_VEL
LIN {X 0,Y 511.705,Z 376.563,A -85,B 0,C 180,E1 -5476.017,E2 -5476.017} C_VEL
LIN {X 0,Y 511.413,Z 389.958,A -85,B 0,C 180,E1 -5476.363,E2 -5476.363} C_VEL
LIN {X 0,Y 511.07,Z 403.324,A -85,B 0,C 180,E1 -5476.885,E2 -5476.885} C_VEL
LIN {X 0,Y 510.832,Z 414.928,A -85,B 0,C 180,E1 -5477.509,E2 -5477.509} C_VEL
LIN {X 0,Y 510.456,Z 426.196,A -85,B 0,C 180,E1 -5478.283,E2 -5478.283} C_VEL
LIN {X 0,Y 510.2,Z 436.692,A -85,B 0,C 180,E1 -5479.182,E2 -5479.182} C_VEL
LIN {X 0,Y 509.86,Z 445.27,A -85,B 0,C 180,E1 -5480.078,E2 -5480.078} C_VEL
LIN {X 0,Y 509.656,Z 453.193,A -85,B 0,C 180,E1 -5481.075,E2 -5481.075} C_VEL
LIN {X 0,Y 509.436,Z 460.931,A -85,B 0,C 180,E1 -5482.269,E2 -5482.269} C_VEL
LIN {X 0,Y 509.309,Z 468.067,A -85,B 0,C 180,E1 -5483.661,E2 -5483.661} C_VEL
LIN {X 0,Y 509.242,Z 472.817,A -85,B 0,C 180,E1 -5484.852,E2 -5484.852} C_VEL
LIN {X 0,Y 509.247,Z 476.449,A -85,B 0,C 180,E1 -5486.042,E2 -5486.042} C_VEL
LIN {X 0,Y 509.201,Z 478.321,A -85,B 0,C 180,E1 -5486.834,E2 -5486.834} C_VEL
LIN {X 0,Y 509.19,Z 479.727,A -85,B 0,C 180,E1 -5487.626,E2 -5487.626} C_VEL
LIN {X 0,Y 509.08,Z 481.34,A -85,B 0,C 180,E1 -5489.208,E2 -5489.208} C_VEL
LIN {X 0,Y 509.078,Z 481.56,A -85,B 0,C 180,E1 -5489.999,E2 -5489.999} C_VEL
LIN {X 0,Y 509.112,Z 480.74,A -85,B 0,C 180,E1 -5491.581,E2 -5491.581} C_VEL
LIN {X 0,Y 509.19,Z 479.747,A -85,B 0,C 180,E1 -5492.372,E2 -5492.372} C_VEL
LIN {X 0,Y 509.2,Z 478.348,A -85,B 0,C 180,E1 -5493.163,E2 -5493.163} C_VEL
LIN {X 0,Y 509.203,Z 475.403,A -85,B 0,C 180,E1 -5494.352,E2 -5494.352} C_VEL
LIN {X 0,Y 509.283,Z 471.418,A -85,B 0,C 180,E1 -5495.541,E2 -5495.541} C_VEL
LIN {X 0,Y 509.329,Z 465.385,A -85,B 0,C 180,E1 -5496.913,E2 -5496.913} C_VEL
LIN {X 0,Y 509.512,Z 458.585,A -85,B 0,C 180,E1 -5498.126,E2 -5498.126} C_VEL
LIN {X 0,Y 509.73,Z 450.275,A -85,B 0,C 180,E1 -5499.321,E2 -5499.321} C_VEL
LIN {X 0,Y 509.965,Z 441.757,A -85,B 0,C 180,E1 -5500.318,E2 -5500.318} C_VEL
LIN {X 0,Y 510.348,Z 431.24,A -85,B 0,C 180,E1 -5501.315,E2 -5501.315} C_VEL
LIN {X 0,Y 510.668,Z 420.894,A -85,B 0,C 180,E1 -5502.108,E2 -5502.108} C_VEL
LIN {X 0,Y 510.979,Z 409.432,A -85,B 0,C 180,E1 -5502.811,E2 -5502.811} C_VEL
LIN {X 0,Y 511.253,Z 397.724,A -85,B 0,C 180,E1 -5503.36,E2 -5503.36} C_VEL
LIN {X 0,Y 511.558,Z 384.244,A -85,B 0,C 180,E1 -5503.807,E2 -5503.807} C_VEL
LIN {X 0,Y 511.793,Z 370.885,A -85,B 0,C 180,E1 -5504.08,E2 -5504.08} C_VEL
LIN {X 0,Y 512.008,Z 280.518,A -85,B 0,C 180,E1 -5505.36,E2 -5505.36} C_VEL
LIN {X 0,Y 510.237,Z 268.37,A -85,B 0,C 180,E1 -5505.589,E2 -5505.589} C_VEL
LIN {X 0,Y 510.729,Z 248.23,A -85,B 0,C 180,E1 -5508.656,E2 -5508.656} C_VEL
LIN {X 0,Y 511.221,Z 227.939,A -85,B 0,C 180,E1 -5511.785,E2 -5511.785} C_VEL
LIN {X 0,Y 511.618,Z 215.723,A -85,B 0,C 180,E1 -5513.687,E2 -5513.687} C_VEL
LIN {X 0,Y 509.877,Z 205.973,A -85,B 0,C 180,E1 -5515.347,E2 -5515.347} C_VEL
LIN {X 0,Y 509.885,Z 205.976,A -85,B 0,C 180,E1 -5518.097,E2 -5518.097} C_VEL
LIN {X 0,Y 509.83,Z 205.974,A -85,B 0,C 180,E1 -5521.276,E2 -5521.276} C_VEL
LIN {X 0,Y 509.843,Z 205.978,A -85,B 0,C 180,E1 -5524.2,E2 -5524.2} C_VEL
LIN {X 0,Y 509.797,Z 205.979,A -85,B 0,C 180,E1 -5527.337,E2 -5527.337} C_VEL
LIN {X 0,Y 509.813,Z 205.978,A -85,B 0,C 180,E1 -5530.378,E2 -5530.378} C_VEL
LIN {X 0,Y 509.795,Z 205.978,A -85,B 0,C 180,E1 -5533.058,E2 -5533.058} C_VEL
LIN {X 0,Y 509.801,Z 205.985,A -85,B 0,C 180,E1 -5535.788,E2 -5535.788} C_VEL
LIN {X 0,Y 509.84,Z 205.972,A -85,B 0,C 180,E1 -5538.573,E2 -5538.573} C_VEL
LIN {X 0,Y 509.82,Z 205.983,A -85,B 0,C 180,E1 -5541.782,E2 -5541.782} C_VEL
LIN {X 0,Y 509.807,Z 205.976,A -85,B 0,C 180,E1 -5544.62,E2 -5544.62} C_VEL
LIN {X 0,Y 509.825,Z 205.981,A -85,B 0,C 180,E1 -5547.478,E2 -5547.478} C_VEL
LIN {X 0,Y 509.839,Z 205.973,A -85,B 0,C 180,E1 -5550.266,E2 -5550.266} C_VEL
LIN {X 0,Y 509.842,Z 205.973,A -85,B 0,C 180,E1 -5552.942,E2 -5552.942} C_VEL
LIN {X 0,Y 509.846,Z 205.979,A -85,B 0,C 180,E1 -5555.573,E2 -5555.573} C_VEL
LIN {X 0,Y 509.805,Z 205.977,A -85,B 0,C 180,E1 -5558.148,E2 -5558.148} C_VEL
LIN {X 0,Y 509.816,Z 205.976,A -85,B 0,C 180,E1 -5560.679,E2 -5560.679} C_VEL
LIN {X 0,Y 509.85,Z 205.977,A -85,B 0,C 180,E1 -5563.173,E2 -5563.173} C_VEL
LIN {X 0,Y 509.822,Z 205.979,A -85,B 0,C 180,E1 -5565.633,E2 -5565.633} C_VEL
LIN {X 0,Y 509.889,Z 205.966,A -85,B 0,C 180,E1 -5568.099,E2 -5568.099} C_VEL
LIN {X 0,Y 509.894,Z 205.974,A -85,B 0,C 180,E1 -5571.279,E2 -5571.279} C_VEL
LIN {X 0,Y 509.936,Z 205.963,A -85,B 0,C 180,E1 -5573.67,E2 -5573.67} C_VEL
LIN {X 0,Y 509.907,Z 205.968,A -85,B 0,C 180,E1 -5576.839,E2 -5576.839} C_VEL
LIN {X 0,Y 510.012,Z 205.958,A -85,B 0,C 180,E1 -5579.21,E2 -5579.21} C_VEL
LIN {X 0,Y 509.88,Z 205.969,A -85,B 0,C 180,E1 -5581.579,E2 -5581.579} C_VEL
LIN {X 0,Y 509.905,Z 205.971,A -85,B 0,C 180,E1 -5583.16,E2 -5583.16} C_VEL
LIN {X 0,Y 509.896,Z 205.966,A -85,B 0,C 180,E1 -5586.33,E2 -5586.33} C_VEL
LIN {X 0,Y 509.863,Z 205.975,A -85,B 0,C 180,E1 -5588.721,E2 -5588.721} C_VEL
LIN {X 0,Y 509.896,Z 205.965,A -85,B 0,C 180,E1 -5591.932,E2 -5591.932} C_VEL
LIN {X 0,Y 509.839,Z 205.975,A -85,B 0,C 180,E1 -5595.243,E2 -5595.243} C_VEL
LIN {X 0,Y 509.835,Z 205.973,A -85,B 0,C 180,E1 -5598.003,E2 -5598.003} C_VEL
LIN {X 0,Y 509.805,Z 205.981,A -85,B 0,C 180,E1 -5601.003,E2 -5601.003} C_VEL
LIN {X 0,Y 509.799,Z 205.977,A -85,B 0,C 180,E1 -5603.565,E2 -5603.565} C_VEL
LIN {X 0,Y 509.864,Z 205.974,A -85,B 0,C 180,E1 -5606.381,E2 -5606.381} C_VEL
LIN {X 0,Y 509.831,Z 205.978,A -85,B 0,C 180,E1 -5608.847,E2 -5608.847} C_VEL
LIN {X 0,Y 509.779,Z 205.98,A -85,B 0,C 180,E1 -5611.593,E2 -5611.593} C_VEL
LIN {X 0,Y 509.81,Z 205.984,A -85,B 0,C 180,E1 -5614.416,E2 -5614.416} C_VEL
LIN {X 0,Y 509.778,Z 205.98,A -85,B 0,C 180,E1 -5617.344,E2 -5617.344} C_VEL
LIN {X 0,Y 509.801,Z 205.986,A -85,B 0,C 180,E1 -5620.385,E2 -5620.385} C_VEL
LIN {X 0,Y 509.788,Z 205.979,A -85,B 0,C 180,E1 -5623.066,E2 -5623.066} C_VEL
LIN {X 0,Y 509.789,Z 205.981,A -85,B 0,C 180,E1 -5625.797,E2 -5625.797} C_VEL
LIN {X 0,Y 509.828,Z 205.978,A -85,B 0,C 180,E1 -5628.578,E2 -5628.578} C_VEL
LIN {X 0,Y 509.824,Z 205.977,A -85,B 0,C 180,E1 -5631.79,E2 -5631.79} C_VEL
LIN {X 0,Y 509.804,Z 205.978,A -85,B 0,C 180,E1 -5633.769,E2 -5633.769} C_VEL
LIN {X 0,Y 509.14,Z 206.064,A -85,B 0,C 180,E1 -5634.429,E2 -5634.429} C_VEL
LIN {X 0,Y 506.323,Z 206.411,A -85,B 0,C 180,E1 -5635.501,E2 -5635.501} C_VEL
LIN {X 0,Y 503.93,Z 206.713,A -85,B 0,C 180,E1 -5636.364,E2 -5636.364} C_VEL
LIN {X 0,Y 502.881,Z 206.839,A -85,B 0,C 180,E1 -5637.031,E2 -5637.031} C_VEL
LIN {X 0,Y 502.784,Z 206.851,A -85,B 0,C 180,E1 -5637.256,E2 -5637.256} C_VEL
LIN {X 0,Y 502.796,Z 206.858,A -85,B 0,C 180,E1 -5640.068,E2 -5640.068} C_VEL
LIN {X 0,Y 502.813,Z 206.849,A -85,B 0,C 180,E1 -5642.536,E2 -5642.536} C_VEL
LIN {X 0,Y 502.789,Z 206.852,A -85,B 0,C 180,E1 -5645.308,E2 -5645.308} C_VEL
LIN {X 0,Y 502.767,Z 206.861,A -85,B 0,C 180,E1 -5647.83,E2 -5647.83} C_VEL
LIN {X 0,Y 502.808,Z 206.85,A -85,B 0,C 180,E1 -5650.403,E2 -5650.403} C_VEL
LIN {X 0,Y 502.799,Z 206.849,A -85,B 0,C 180,E1 -5652.934,E2 -5652.934} C_VEL
LIN {X 0,Y 502.826,Z 206.85,A -85,B 0,C 180,E1 -5655.431,E2 -5655.431} C_VEL
LIN {X 0,Y 502.871,Z 206.84,A -85,B 0,C 180,E1 -5658.719,E2 -5658.719} C_VEL
LIN {X 0,Y 502.876,Z 206.847,A -85,B 0,C 180,E1 -5661.968,E2 -5661.968} C_VEL
LIN {X 0,Y 502.923,Z 206.838,A -85,B 0,C 180,E1 -5664.388,E2 -5664.388} C_VEL
LIN {X 0,Y 502.85,Z 206.939,A -85,B 0,C 180,E1 -5665.769,E2 -5665.769} C_VEL
LIN {X 0,Y 503.446,Z 212.046,A -85,B 0,C 180,E1 -5666.801,E2 -5666.801} C_VEL
LIN {X 0,Y 503.309,Z 224.625,A -85,B 0,C 180,E1 -5669.251,E2 -5669.251} C_VEL
LIN {X 0,Y 505.499,Z 236.457,A -85,B 0,C 180,E1 -5669.504,E2 -5669.504} C_VEL
LIN {X 0,Y 504.895,Z 331.172,A -85,B 0,C 180,E1 -5670.874,E2 -5670.874} C_VEL
LIN {X 0,Y 504.689,Z 344.371,A -85,B 0,C 180,E1 -5671.223,E2 -5671.223} C_VEL
LIN {X 0,Y 504.455,Z 357.53,A -85,B 0,C 180,E1 -5671.748,E2 -5671.748} C_VEL
LIN {X 0,Y 504.126,Z 369.437,A -85,B 0,C 180,E1 -5672.398,E2 -5672.398} C_VEL
LIN {X 0,Y 503.702,Z 380.832,A -85,B 0,C 180,E1 -5673.2,E2 -5673.2} C_VEL
LIN {X 0,Y 503.382,Z 391.08,A -85,B 0,C 180,E1 -5674.104,E2 -5674.104} C_VEL
LIN {X 0,Y 503.061,Z 399.492,A -85,B 0,C 180,E1 -5675.01,E2 -5675.01} C_VEL
LIN {X 0,Y 502.84,Z 407.245,A -85,B 0,C 180,E1 -5676.018,E2 -5676.018} C_VEL
LIN {X 0,Y 502.614,Z 414.843,A -85,B 0,C 180,E1 -5677.23,E2 -5677.23} C_VEL
LIN {X 0,Y 502.423,Z 420.969,A -85,B 0,C 180,E1 -5678.447,E2 -5678.447} C_VEL
LIN {X 0,Y 502.252,Z 425.845,A -85,B 0,C 180,E1 -5679.667,E2 -5679.667} C_VEL
LIN {X 0,Y 502.181,Z 429.595,A -85,B 0,C 180,E1 -5680.891,E2 -5680.891} C_VEL
LIN {X 0,Y 502.097,Z 432.322,A -85,B 0,C 180,E1 -5682.12,E2 -5682.12} C_VEL
LIN {X 0,Y 502.038,Z 433.608,A -85,B 0,C 180,E1 -5682.943,E2 -5682.943} C_VEL
LIN {X 0,Y 502.035,Z 434.479,A -85,B 0,C 180,E1 -5683.768,E2 -5683.768} C_VEL
LIN {X 0,Y 502.049,Z 434.978,A -85,B 0,C 180,E1 -5685.006,E2 -5685.006} C_VEL
LIN {X 0,Y 502.011,Z 434.53,A -85,B 0,C 180,E1 -5686.26,E2 -5686.26} C_VEL
LIN {X 0,Y 502.053,Z 433.692,A -85,B 0,C 180,E1 -5687.096,E2 -5687.096} C_VEL
LIN {X 0,Y 502.092,Z 432.404,A -85,B 0,C 180,E1 -5687.935,E2 -5687.935} C_VEL
LIN {X 0,Y 502.165,Z 429.621,A -85,B 0,C 180,E1 -5689.201,E2 -5689.201} C_VEL
LIN {X 0,Y 502.265,Z 425.702,A -85,B 0,C 180,E1 -5690.476,E2 -5690.476} C_VEL
LIN {X 0,Y 502.403,Z 420.512,A -85,B 0,C 180,E1 -5691.758,E2 -5691.758} C_VEL
LIN {X 0,Y 502.633,Z 413.849,A -85,B 0,C 180,E1 -5693.048,E2 -5693.048} C_VEL
LIN {X 0,Y 502.911,Z 405.321,A -85,B 0,C 180,E1 -5694.346,E2 -5694.346} C_VEL
LIN {X 0,Y 503.209,Z 396.476,A -85,B 0,C 180,E1 -5695.433,E2 -5695.433} C_VEL
LIN {X 0,Y 503.541,Z 386.599,A -85,B 0,C 180,E1 -5696.415,E2 -5696.415} C_VEL
LIN {X 0,Y 503.917,Z 375.414,A -85,B 0,C 180,E1 -5697.304,E2 -5697.304} C_VEL
LIN {X 0,Y 504.324,Z 363.415,A -85,B 0,C 180,E1 -5698.054,E2 -5698.054} C_VEL
LIN {X 0,Y 504.584,Z 351.546,A -85,B 0,C 180,E1 -5698.614,E2 -5698.614} C_VEL
LIN {X 0,Y 504.774,Z 338.415,A -85,B 0,C 180,E1 -5699.055,E2 -5699.055} C_VEL
LIN {X 0,Y 504.901,Z 325.306,A -85,B 0,C 180,E1 -5699.326,E2 -5699.326} C_VEL
LIN {X 0,Y 505.378,Z 235.218,A -85,B 0,C 180,E1 -5700.618,E2 -5700.618} C_VEL
LIN {X 0,Y 503.271,Z 224.64,A -85,B 0,C 180,E1 -5700.855,E2 -5700.855} C_VEL
LIN {X 0,Y 503.449,Z 212.793,A -85,B 0,C 180,E1 -5703.115,E2 -5703.115} C_VEL
LIN {X 0,Y 503.148,Z 208.422,A -85,B 0,C 180,E1 -5703.966,E2 -5703.966} C_VEL
LIN {X 0,Y 502.879,Z 206.847,A -85,B 0,C 180,E1 -5704.307,E2 -5704.307} C_VEL
LIN {X 0,Y 502.784,Z 206.857,A -85,B 0,C 180,E1 -5707.952,E2 -5707.952} C_VEL
LIN {X 0,Y 502.816,Z 206.848,A -85,B 0,C 180,E1 -5711.064,E2 -5711.064} C_VEL
LIN {X 0,Y 502.768,Z 206.857,A -85,B 0,C 180,E1 -5713.374,E2 -5713.374} C_VEL
LIN {X 0,Y 502.774,Z 206.856,A -85,B 0,C 180,E1 -5715.66,E2 -5715.66} C_VEL
LIN {X 0,Y 502.813,Z 206.853,A -85,B 0,C 180,E1 -5717.863,E2 -5717.863} C_VEL
LIN {X 0,Y 502.79,Z 206.852,A -85,B 0,C 180,E1 -5721.023,E2 -5721.023} C_VEL
LIN {X 0,Y 502.764,Z 206.859,A -85,B 0,C 180,E1 -5724.166,E2 -5724.166} C_VEL
LIN {X 0,Y 502.811,Z 206.848,A -85,B 0,C 180,E1 -5726.992,E2 -5726.992} C_VEL
LIN {X 0,Y 502.806,Z 206.854,A -85,B 0,C 180,E1 -5730.06,E2 -5730.06} C_VEL
LIN {X 0,Y 502.809,Z 206.848,A -85,B 0,C 180,E1 -5732.532,E2 -5732.532} C_VEL
LIN {X 0,Y 502.81,Z 206.848,A -85,B 0,C 180,E1 -5735.295,E2 -5735.295} C_VEL
LIN {X 0,Y 502.793,Z 206.855,A -85,B 0,C 180,E1 -5737.827,E2 -5737.827} C_VEL
LIN {X 0,Y 502.797,Z 206.85,A -85,B 0,C 180,E1 -5740.399,E2 -5740.399} C_VEL
LIN {X 0,Y 502.817,Z 206.846,A -85,B 0,C 180,E1 -5742.931,E2 -5742.931} C_VEL
LIN {X 0,Y 502.82,Z 206.854,A -85,B 0,C 180,E1 -5745.429,E2 -5745.429} C_VEL
LIN {X 0,Y 502.849,Z 206.843,A -85,B 0,C 180,E1 -5748.716,E2 -5748.716} C_VEL
LIN {X 0,Y 502.874,Z 206.839,A -85,B 0,C 180,E1 -5751.966,E2 -5751.966} C_VEL
LIN {X 0,Y 502.918,Z 206.834,A -85,B 0,C 180,E1 -5754.387,E2 -5754.387} C_VEL
LIN {X 0,Y 502.99,Z 206.829,A -85,B 0,C 180,E1 -5757.598,E2 -5757.598} C_VEL
LIN {X 0,Y 502.987,Z 206.824,A -85,B 0,C 180,E1 -5760,E2 -5760} C_VEL
LIN {X 0,Y 502.988,Z 206.823,A -85,B 0,C 180,E1 -5762.403,E2 -5762.403} C_VEL
LIN {X 0,Y 502.899,Z 206.835,A -85,B 0,C 180,E1 -5765.614,E2 -5765.614} C_VEL
LIN {X 0,Y 502.848,Z 206.842,A -85,B 0,C 180,E1 -5768.034,E2 -5768.034} C_VEL
LIN {X 0,Y 502.869,Z 206.844,A -85,B 0,C 180,E1 -5771.284,E2 -5771.284} C_VEL
LIN {X 0,Y 502.811,Z 206.849,A -85,B 0,C 180,E1 -5774.572,E2 -5774.572} C_VEL
LIN {X 0,Y 502.791,Z 206.849,A -85,B 0,C 180,E1 -5777.91,E2 -5777.91} C_VEL
LIN {X 0,Y 502.802,Z 206.852,A -85,B 0,C 180,E1 -5780.538,E2 -5780.538} C_VEL
LIN {X 0,Y 502.758,Z 206.857,A -85,B 0,C 180,E1 -5783.042,E2 -5783.042} C_VEL
LIN {X 0,Y 502.758,Z 206.855,A -85,B 0,C 180,E1 -5785.68,E2 -5785.68} C_VEL
LIN {X 0,Y 502.771,Z 206.856,A -85,B 0,C 180,E1 -5788.377,E2 -5788.377} C_VEL
LIN {X 0,Y 502.77,Z 206.854,A -85,B 0,C 180,E1 -5791.145,E2 -5791.145} C_VEL
LIN {X 0,Y 502.766,Z 206.856,A -85,B 0,C 180,E1 -5793.997,E2 -5793.997} C_VEL
LIN {X 0,Y 502.744,Z 206.856,A -85,B 0,C 180,E1 -5797.177,E2 -5797.177} C_VEL
LIN {X 0,Y 502.766,Z 206.858,A -85,B 0,C 180,E1 -5800.018,E2 -5800.018} C_VEL
LIN {X 0,Y 502.788,Z 206.851,A -85,B 0,C 180,E1 -5802.201,E2 -5802.201} C_VEL
LIN {X 0,Y 502.772,Z 206.853,A -85,B 0,C 180,E1 -5805.472,E2 -5805.472} C_VEL
LIN {X 0,Y 502.784,Z 206.856,A -85,B 0,C 180,E1 -5807.862,E2 -5807.862} C_VEL
LIN {X 0,Y 502.784,Z 206.853,A -85,B 0,C 180,E1 -5811.025,E2 -5811.025} C_VEL
LIN {X 0,Y 502.77,Z 206.862,A -85,B 0,C 180,E1 -5814.17,E2 -5814.17} C_VEL
LIN {X 0,Y 502.828,Z 206.848,A -85,B 0,C 180,E1 -5816.995,E2 -5816.995} C_VEL
LIN {X 0,Y 502.812,Z 206.856,A -85,B 0,C 180,E1 -5820.066,E2 -5820.066} C_VEL
LIN {X 0,Y 502.843,Z 206.852,A -85,B 0,C 180,E1 -5823.445,E2 -5823.445} C_VEL
LIN {X 0,Y 502.85,Z 207.005,A -85,B 0,C 180,E1 -5824.548,E2 -5824.548} C_VEL
LIN {X 0,Y 504.597,Z 216.542,A -85,B 0,C 180,E1 -5826.178,E2 -5826.178} C_VEL
LIN {X 0,Y 504.094,Z 234.938,A -85,B 0,C 180,E1 -5829.085,E2 -5829.085} C_VEL
LIN {X 0,Y 503.565,Z 254.444,A -85,B 0,C 180,E1 -5832.119,E2 -5832.119} C_VEL
LIN {X 0,Y 503.208,Z 267.844,A -85,B 0,C 180,E1 -5834.179,E2 -5834.179} C_VEL
LIN {X 0,Y 505.323,Z 282.397,A -85,B 0,C 180,E1 -5834.463,E2 -5834.463} C_VEL
LIN {X 0,Y 504.831,Z 376.255,A -85,B 0,C 180,E1 -5835.822,E2 -5835.822} C_VEL
LIN {X 0,Y 504.518,Z 389.626,A -85,B 0,C 180,E1 -5836.173,E2 -5836.173} C_VEL
LIN {X 0,Y 504.156,Z 402.979,A -85,B 0,C 180,E1 -5836.702,E2 -5836.702} C_VEL
LIN {X 0,Y 503.841,Z 415.387,A -85,B 0,C 180,E1 -5837.386,E2 -5837.386} C_VEL
LIN {X 0,Y 503.437,Z 427.145,A -85,B 0,C 180,E1 -5838.219,E2 -5838.219} C_VEL
LIN {X 0,Y 503.156,Z 437.399,A -85,B 0,C 180,E1 -5839.131,E2 -5839.131} C_VEL
LIN {X 0,Y 502.788,Z 446.618,A -85,B 0,C 180,E1 -5840.14,E2 -5840.14} C_VEL
LIN {X 0,Y 502.535,Z 455.607,A -85,B 0,C 180,E1 -5841.353,E2 -5841.353} C_VEL
LIN {X 0,Y 502.333,Z 462.845,A -85,B 0,C 180,E1 -5842.564,E2 -5842.564} C_VEL
LIN {X 0,Y 502.237,Z 467.732,A -85,B 0,C 180,E1 -5843.572,E2 -5843.572} C_VEL
LIN {X 0,Y 502.171,Z 472.484,A -85,B 0,C 180,E1 -5844.78,E2 -5844.78} C_VEL
LIN {X 0,Y 502.141,Z 476.117,A -85,B 0,C 180,E1 -5845.986,E2 -5845.986} C_VEL
LIN {X 0,Y 502.121,Z 477.992,A -85,B 0,C 180,E1 -5846.789,E2 -5846.789} C_VEL
LIN {X 0,Y 502.121,Z 479.399,A -85,B 0,C 180,E1 -5847.592,E2 -5847.592} C_VEL
LIN {X 0,Y 501.996,Z 481.013,A -85,B 0,C 180,E1 -5849.197,E2 -5849.197} C_VEL
LIN {X 0,Y 501.992,Z 481.234,A -85,B 0,C 180,E1 -5849.999,E2 -5849.999} C_VEL
LIN {X 0,Y 502.036,Z 480.415,A -85,B 0,C 180,E1 -5851.603,E2 -5851.603} C_VEL
LIN {X 0,Y 502.121,Z 479.422,A -85,B 0,C 180,E1 -5852.405,E2 -5852.405} C_VEL
LIN {X 0,Y 502.12,Z 478.022,A -85,B 0,C 180,E1 -5853.208,E2 -5853.208} C_VEL
LIN {X 0,Y 502.101,Z 475.076,A -85,B 0,C 180,E1 -5854.413,E2 -5854.413} C_VEL
LIN {X 0,Y 502.199,Z 471.091,A -85,B 0,C 180,E1 -5855.62,E2 -5855.62} C_VEL
LIN {X 0,Y 502.271,Z 465.058,A -85,B 0,C 180,E1 -5857.01,E2 -5857.01} C_VEL
LIN {X 0,Y 502.459,Z 458.257,A -85,B 0,C 180,E1 -5858.241,E2 -5858.241} C_VEL
LIN {X 0,Y 502.696,Z 449.945,A -85,B 0,C 180,E1 -5859.453,E2 -5859.453} C_VEL
LIN {X 0,Y 502.95,Z 441.425,A -85,B 0,C 180,E1 -5860.464,E2 -5860.464} C_VEL
LIN {X 0,Y 503.367,Z 430.906,A -85,B 0,C 180,E1 -5861.474,E2 -5861.474} C_VEL
LIN {X 0,Y 503.681,Z 420.556,A -85,B 0,C 180,E1 -5862.279,E2 -5862.279} C_VEL
LIN {X 0,Y 504.024,Z 409.091,A -85,B 0,C 180,E1 -5862.991,E2 -5862.991} C_VEL
LIN {X 0,Y 504.31,Z 397.375,A -85,B 0,C 180,E1 -5863.547,E2 -5863.547} C_VEL
LIN {X 0,Y 504.665,Z 383.888,A -85,B 0,C 180,E1 -5864,E2 -5864} C_VEL
LIN {X 0,Y 504.912,Z 370.492,A -85,B 0,C 180,E1 -5864.276,E2 -5864.276} C_VEL
LIN {X 0,Y 505.189,Z 281.496,A -85,B 0,C 180,E1 -5865.553,E2 -5865.553} C_VEL
LIN {X 0,Y 503.228,Z 267.999,A -85,B 0,C 180,E1 -5865.818,E2 -5865.818} C_VEL
LIN {X 0,Y 503.738,Z 249.24,A -85,B 0,C 180,E1 -5868.713,E2 -5868.713} C_VEL
LIN {X 0,Y 504.264,Z 228.921,A -85,B 0,C 180,E1 -5871.886,E2 -5871.886} C_VEL
LIN {X 0,Y 504.635,Z 216.68,A -85,B 0,C 180,E1 -5873.817,E2 -5873.817} C_VEL
LIN {X 0,Y 502.849,Z 206.85,A -85,B 0,C 180,E1 -5875.505,E2 -5875.505} C_VEL
LIN {X 0,Y 502.827,Z 206.854,A -85,B 0,C 180,E1 -5878.369,E2 -5878.369} C_VEL
LIN {X 0,Y 502.777,Z 206.853,A -85,B 0,C 180,E1 -5881.495,E2 -5881.495} C_VEL
LIN {X 0,Y 502.788,Z 206.854,A -85,B 0,C 180,E1 -5884.441,E2 -5884.441} C_VEL
LIN {X 0,Y 502.759,Z 206.854,A -85,B 0,C 180,E1 -5887.174,E2 -5887.174} C_VEL
LIN {X 0,Y 502.763,Z 206.861,A -85,B 0,C 180,E1 -5890.011,E2 -5890.011} C_VEL
LIN {X 0,Y 502.776,Z 206.856,A -85,B 0,C 180,E1 -5892.195,E2 -5892.195} C_VEL
LIN {X 0,Y 502.771,Z 206.856,A -85,B 0,C 180,E1 -5895.464,E2 -5895.464} C_VEL
LIN {X 0,Y 502.807,Z 206.856,A -85,B 0,C 180,E1 -5897.861,E2 -5897.861} C_VEL
LIN {X 0,Y 502.787,Z 206.851,A -85,B 0,C 180,E1 -5901.022,E2 -5901.022} C_VEL
LIN {X 0,Y 502.747,Z 206.858,A -85,B 0,C 180,E1 -5904.164,E2 -5904.164} C_VEL
LIN {X 0,Y 502.792,Z 206.851,A -85,B 0,C 180,E1 -5906.99,E2 -5906.99} C_VEL
LIN {X 0,Y 502.788,Z 206.853,A -85,B 0,C 180,E1 -5910.058,E2 -5910.058} C_VEL
LIN {X 0,Y 502.791,Z 206.85,A -85,B 0,C 180,E1 -5912.53,E2 -5912.53} C_VEL
LIN {X 0,Y 502.791,Z 206.856,A -85,B 0,C 180,E1 -5915.293,E2 -5915.293} C_VEL
LIN {X 0,Y 502.772,Z 206.856,A -85,B 0,C 180,E1 -5917.826,E2 -5917.826} C_VEL
LIN {X 0,Y 502.776,Z 206.852,A -85,B 0,C 180,E1 -5920.398,E2 -5920.398} C_VEL
LIN {X 0,Y 502.796,Z 206.852,A -85,B 0,C 180,E1 -5922.93,E2 -5922.93} C_VEL
LIN {X 0,Y 502.8,Z 206.856,A -85,B 0,C 180,E1 -5925.428,E2 -5925.428} C_VEL
LIN {X 0,Y 502.848,Z 206.845,A -85,B 0,C 180,E1 -5928.716,E2 -5928.716} C_VEL
LIN {X 0,Y 502.863,Z 206.842,A -85,B 0,C 180,E1 -5931.966,E2 -5931.966} C_VEL
LIN {X 0,Y 502.909,Z 206.836,A -85,B 0,C 180,E1 -5934.386,E2 -5934.386} C_VEL
LIN {X 0,Y 502.968,Z 206.831,A -85,B 0,C 180,E1 -5937.597,E2 -5937.597} C_VEL
LIN {X 0,Y 502.965,Z 206.828,A -85,B 0,C 180,E1 -5940,E2 -5940} C_VEL
LIN {X 0,Y 502.967,Z 206.829,A -85,B 0,C 180,E1 -5942.402,E2 -5942.402} C_VEL
LIN {X 0,Y 502.886,Z 206.839,A -85,B 0,C 180,E1 -5945.614,E2 -5945.614} C_VEL
LIN {X 0,Y 502.846,Z 206.843,A -85,B 0,C 180,E1 -5948.034,E2 -5948.034} C_VEL
LIN {X 0,Y 502.846,Z 206.847,A -85,B 0,C 180,E1 -5951.284,E2 -5951.284} C_VEL
LIN {X 0,Y 502.789,Z 206.856,A -85,B 0,C 180,E1 -5954.572,E2 -5954.572} C_VEL
LIN {X 0,Y 502.81,Z 206.848,A -85,B 0,C 180,E1 -5957.909,E2 -5957.909} C_VEL
LIN {X 0,Y 502.778,Z 206.858,A -85,B 0,C 180,E1 -5960.538,E2 -5960.538} C_VEL
LIN {X 0,Y 502.755,Z 206.858,A -85,B 0,C 180,E1 -5963.042,E2 -5963.042} C_VEL
LIN {X 0,Y 502.792,Z 206.85,A -85,B 0,C 180,E1 -5965.678,E2 -5965.678} C_VEL
LIN {X 0,Y 502.794,Z 206.855,A -85,B 0,C 180,E1 -5968.375,E2 -5968.375} C_VEL
LIN {X 0,Y 502.751,Z 206.855,A -85,B 0,C 180,E1 -5971.502,E2 -5971.502} C_VEL
LIN {X 0,Y 502.763,Z 206.862,A -85,B 0,C 180,E1 -5974.447,E2 -5974.447} C_VEL
LIN {X 0,Y 502.741,Z 206.857,A -85,B 0,C 180,E1 -5977.181,E2 -5977.181} C_VEL
LIN {X 0,Y 502.75,Z 206.859,A -85,B 0,C 180,E1 -5980.018,E2 -5980.018} C_VEL
LIN {X 0,Y 502.767,Z 206.86,A -85,B 0,C 180,E1 -5982.203,E2 -5982.203} C_VEL
LIN {X 0,Y 502.752,Z 206.855,A -85,B 0,C 180,E1 -5985.474,E2 -5985.474} C_VEL
LIN {X 0,Y 502.791,Z 206.851,A -85,B 0,C 180,E1 -5988.938,E2 -5988.938} C_VEL
LIN {X 0,Y 502.767,Z 206.86,A -85,B 0,C 180,E1 -5992.05,E2 -5992.05} C_VEL
LIN {X 0,Y 502.784,Z 206.851,A -85,B 0,C 180,E1 -5995.038,E2 -5995.038} C_VEL
LIN {X 0,Y 502.784,Z 206.851,A -85,B 0,C 180,E1 -5997.256,E2 -5997.256} C_VEL
LIN {X 0,Y 502.084,Z 206.945,A -85,B 0,C 180,E1 -5997.925,E2 -5997.925} C_VEL
LIN {X 0,Y 499.22,Z 207.3,A -85,B 0,C 180,E1 -5999.011,E2 -5999.011} C_VEL
LIN {X 0,Y 496.827,Z 207.599,A -85,B 0,C 180,E1 -5999.886,E2 -5999.886} C_VEL
LIN {X 0,Y 495.811,Z 207.722,A -85,B 0,C 180,E1 -6000.562,E2 -6000.562} C_VEL
LIN {X 0,Y 495.734,Z 207.73,A -85,B 0,C 180,E1 -6000.79,E2 -6000.79} C_VEL
LIN {X 0,Y 495.765,Z 207.734,A -85,B 0,C 180,E1 -6003.935,E2 -6003.935} C_VEL
LIN {X 0,Y 495.746,Z 207.728,A -85,B 0,C 180,E1 -6007.143,E2 -6007.143} C_VEL
LIN {X 0,Y 495.756,Z 207.732,A -85,B 0,C 180,E1 -6010.112,E2 -6010.112} C_VEL
LIN {X 0,Y 495.745,Z 207.728,A -85,B 0,C 180,E1 -6012.683,E2 -6012.683} C_VEL
LIN {X 0,Y 495.774,Z 207.726,A -85,B 0,C 180,E1 -6015.22,E2 -6015.22} C_VEL
LIN {X 0,Y 495.846,Z 207.716,A -85,B 0,C 180,E1 -6018.557,E2 -6018.557} C_VEL
LIN {X 0,Y 495.833,Z 207.726,A -85,B 0,C 180,E1 -6021.854,E2 -6021.854} C_VEL
LIN {X 0,Y 495.878,Z 207.716,A -85,B 0,C 180,E1 -6024.308,E2 -6024.308} C_VEL
LIN {X 0,Y 495.83,Z 207.762,A -85,B 0,C 180,E1 -6025.632,E2 -6025.632} C_VEL
LIN {X 0,Y 496.457,Z 213.299,A -85,B 0,C 180,E1 -6026.756,E2 -6026.756} C_VEL
LIN {X 0,Y 496.33,Z 224.922,A -85,B 0,C 180,E1 -6029.038,E2 -6029.038} C_VEL
LIN {X 0,Y 498.665,Z 237.114,A -85,B 0,C 180,E1 -6029.295,E2 -6029.295} C_VEL
LIN {X 0,Y 498.015,Z 331.694,A -85,B 0,C 180,E1 -6030.684,E2 -6030.684} C_VEL
LIN {X 0,Y 497.798,Z 344.819,A -85,B 0,C 180,E1 -6031.038,E2 -6031.038} C_VEL
LIN {X 0,Y 497.564,Z 357.934,A -85,B 0,C 180,E1 -6031.569,E2 -6031.569} C_VEL
LIN {X 0,Y 497.204,Z 369.822,A -85,B 0,C 180,E1 -6032.229,E2 -6032.229} C_VEL
LIN {X 0,Y 496.753,Z 381.208,A -85,B 0,C 180,E1 -6033.042,E2 -6033.042} C_VEL
LIN {X 0,Y 496.403,Z 391.451,A -85,B 0,C 180,E1 -6033.959,E2 -6033.959} C_VEL
LIN {X 0,Y 496.058,Z 399.861,A -85,B 0,C 180,E1 -6034.877,E2 -6034.877} C_VEL
LIN {X 0,Y 495.841,Z 407.605,A -85,B 0,C 180,E1 -6035.899,E2 -6035.899} C_VEL
LIN {X 0,Y 495.625,Z 414.355,A -85,B 0,C 180,E1 -6036.974,E2 -6036.974} C_VEL
LIN {X 0,Y 495.415,Z 420.418,A -85,B 0,C 180,E1 -6038.156,E2 -6038.156} C_VEL
LIN {X 0,Y 495.23,Z 425.478,A -85,B 0,C 180,E1 -6039.393,E2 -6039.393} C_VEL
LIN {X 0,Y 495.131,Z 429.403,A -85,B 0,C 180,E1 -6040.634,E2 -6040.634} C_VEL
LIN {X 0,Y 495.082,Z 431.772,A -85,B 0,C 180,E1 -6041.623,E2 -6041.623} C_VEL
LIN {X 0,Y 494.954,Z 434.211,A -85,B 0,C 180,E1 -6043.132,E2 -6043.132} C_VEL
LIN {X 0,Y 494.942,Z 434.937,A -85,B 0,C 180,E1 -6043.969,E2 -6043.969} C_VEL
LIN {X 0,Y 494.962,Z 435.305,A -85,B 0,C 180,E1 -6045.087,E2 -6045.087} C_VEL
LIN {X 0,Y 494.923,Z 434.674,A -85,B 0,C 180,E1 -6046.499,E2 -6046.499} C_VEL
LIN {X 0,Y 495.012,Z 432.751,A -85,B 0,C 180,E1 -6047.967,E2 -6047.967} C_VEL
LIN {X 0,Y 495.117,Z 429.372,A -85,B 0,C 180,E1 -6049.485,E2 -6049.485} C_VEL
LIN {X 0,Y 495.238,Z 425.253,A -85,B 0,C 180,E1 -6050.779,E2 -6050.779} C_VEL
LIN {X 0,Y 495.422,Z 418.742,A -85,B 0,C 180,E1 -6052.3,E2 -6052.3} C_VEL
LIN {X 0,Y 495.689,Z 411.52,A -85,B 0,C 180,E1 -6053.611,E2 -6053.611} C_VEL
LIN {X 0,Y 496.005,Z 402.95,A -85,B 0,C 180,E1 -6054.843,E2 -6054.843} C_VEL
LIN {X 0,Y 496.367,Z 393.662,A -85,B 0,C 180,E1 -6055.921,E2 -6055.921} C_VEL
LIN {X 0,Y 496.719,Z 383.042,A -85,B 0,C 180,E1 -6056.92,E2 -6056.92} C_VEL
LIN {X 0,Y 497.121,Z 372.864,A -85,B 0,C 180,E1 -6057.683,E2 -6057.683} C_VEL
LIN {X 0,Y 497.482,Z 360.388,A -85,B 0,C 180,E1 -6058.417,E2 -6058.417} C_VEL
LIN {X 0,Y 497.783,Z 347.658,A -85,B 0,C 180,E1 -6058.974,E2 -6058.974} C_VEL
LIN {X 0,Y 497.974,Z 334.221,A -85,B 0,C 180,E1 -6059.368,E2 -6059.368} C_VEL
LIN {X 0,Y 498.172,Z 313.587,A -85,B 0,C 180,E1 -6059.703,E2 -6059.703} C_VEL
LIN {X 0,Y 498.663,Z 236.676,A -85,B 0,C 180,E1 -6060.823,E2 -6060.823} C_VEL
LIN {X 0,Y 496.312,Z 224.905,A -85,B 0,C 180,E1 -6061.096,E2 -6061.096} C_VEL
LIN {X 0,Y 496.483,Z 212.363,A -85,B 0,C 180,E1 -6063.507,E2 -6063.507} C_VEL
LIN {X 0,Y 495.799,Z 207.729,A -85,B 0,C 180,E1 -6064.478,E2 -6064.478} C_VEL
LIN {X 0,Y 495.721,Z 207.734,A -85,B 0,C 180,E1 -6067.56,E2 -6067.56} C_VEL
LIN {X 0,Y 495.769,Z 207.729,A -85,B 0,C 180,E1 -6070.697,E2 -6070.697} C_VEL
LIN {X 0,Y 495.72,Z 207.736,A -85,B 0,C 180,E1 -6073.694,E2 -6073.694} C_VEL
LIN {X 0,Y 495.718,Z 207.74,A -85,B 0,C 180,E1 -6076.303,E2 -6076.303} C_VEL
LIN {X 0,Y 495.762,Z 207.727,A -85,B 0,C 180,E1 -6079.3,E2 -6079.3} C_VEL
LIN {X 0,Y 495.711,Z 207.736,A -85,B 0,C 180,E1 -6082.437,E2 -6082.437} C_VEL
LIN {X 0,Y 495.763,Z 207.726,A -85,B 0,C 180,E1 -6085.456,E2 -6085.456} C_VEL
LIN {X 0,Y 495.736,Z 207.731,A -85,B 0,C 180,E1 -6088.363,E2 -6088.363} C_VEL
LIN {X 0,Y 495.765,Z 207.728,A -85,B 0,C 180,E1 -6091.505,E2 -6091.505} C_VEL
LIN {X 0,Y 495.767,Z 207.73,A -85,B 0,C 180,E1 -6093.931,E2 -6093.931} C_VEL
LIN {X 0,Y 495.762,Z 207.727,A -85,B 0,C 180,E1 -6097.13,E2 -6097.13} C_VEL
LIN {X 0,Y 495.75,Z 207.731,A -85,B 0,C 180,E1 -6100.109,E2 -6100.109} C_VEL
LIN {X 0,Y 495.766,Z 207.723,A -85,B 0,C 180,E1 -6102.681,E2 -6102.681} C_VEL
LIN {X 0,Y 495.764,Z 207.73,A -85,B 0,C 180,E1 -6105.217,E2 -6105.217} C_VEL
LIN {X 0,Y 495.823,Z 207.718,A -85,B 0,C 180,E1 -6108.554,E2 -6108.554} C_VEL
LIN {X 0,Y 495.844,Z 207.716,A -85,B 0,C 180,E1 -6111.852,E2 -6111.852} C_VEL
LIN {X 0,Y 495.876,Z 207.711,A -85,B 0,C 180,E1 -6114.307,E2 -6114.307} C_VEL
LIN {X 0,Y 495.959,Z 207.705,A -85,B 0,C 180,E1 -6117.564,E2 -6117.564} C_VEL
LIN {X 0,Y 495.959,Z 207.699,A -85,B 0,C 180,E1 -6120,E2 -6120} C_VEL
LIN {X 0,Y 495.957,Z 207.699,A -85,B 0,C 180,E1 -6122.437,E2 -6122.437} C_VEL
LIN {X 0,Y 495.855,Z 207.711,A -85,B 0,C 180,E1 -6125.694,E2 -6125.694} C_VEL
LIN {X 0,Y 495.804,Z 207.719,A -85,B 0,C 180,E1 -6128.149,E2 -6128.149} C_VEL
LIN {X 0,Y 495.842,Z 207.717,A -85,B 0,C 180,E1 -6131.446,E2 -6131.446} C_VEL
LIN {X 0,Y 495.757,Z 207.73,A -85,B 0,C 180,E1 -6134.784,E2 -6134.784} C_VEL
LIN {X 0,Y 495.732,Z 207.731,A -85,B 0,C 180,E1 -6137.321,E2 -6137.321} C_VEL
LIN {X 0,Y 495.74,Z 207.727,A -85,B 0,C 180,E1 -6139.892,E2 -6139.892} C_VEL
LIN {X 0,Y 495.73,Z 207.734,A -85,B 0,C 180,E1 -6142.861,E2 -6142.861} C_VEL
LIN {X 0,Y 495.716,Z 207.734,A -85,B 0,C 180,E1 -6146.072,E2 -6146.072} C_VEL
LIN {X 0,Y 495.719,Z 207.738,A -85,B 0,C 180,E1 -6148.818,E2 -6148.818} C_VEL
LIN {X 0,Y 495.731,Z 207.729,A -85,B 0,C 180,E1 -6151.726,E2 -6151.726} C_VEL
LIN {X 0,Y 495.74,Z 207.735,A -85,B 0,C 180,E1 -6154.694,E2 -6154.694} C_VEL
LIN {X 0,Y 495.701,Z 207.733,A -85,B 0,C 180,E1 -6157.565,E2 -6157.565} C_VEL
LIN {X 0,Y 495.737,Z 207.734,A -85,B 0,C 180,E1 -6160.048,E2 -6160.048} C_VEL
LIN {X 0,Y 495.711,Z 207.734,A -85,B 0,C 180,E1 -6162.885,E2 -6162.885} C_VEL
LIN {X 0,Y 495.712,Z 207.737,A -85,B 0,C 180,E1 -6166,E2 -6166} C_VEL
LIN {X 0,Y 495.711,Z 207.735,A -85,B 0,C 180,E1 -6168.713,E2 -6168.713} C_VEL
LIN {X 0,Y 495.736,Z 207.731,A -85,B 0,C 180,E1 -6171.409,E2 -6171.409} C_VEL
LIN {X 0,Y 495.743,Z 207.734,A -85,B 0,C 180,E1 -6174.464,E2 -6174.464} C_VEL
LIN {X 0,Y 495.763,Z 207.73,A -85,B 0,C 180,E1 -6177.407,E2 -6177.407} C_VEL
LIN {X 0,Y 495.76,Z 207.733,A -85,B 0,C 180,E1 -6180.255,E2 -6180.255} C_VEL
LIN {X 0,Y 495.773,Z 207.731,A -85,B 0,C 180,E1 -6183.263,E2 -6183.263} C_VEL
LIN {X 0,Y 495.8,Z 207.794,A -85,B 0,C 180,E1 -6184.329,E2 -6184.329} C_VEL
LIN {X 0,Y 497.638,Z 217.674,A -85,B 0,C 180,E1 -6186.045,E2 -6186.045} C_VEL
LIN {X 0,Y 497.326,Z 231.186,A -85,B 0,C 180,E1 -6188.226,E2 -6188.226} C_VEL
LIN {X 0,Y 496.615,Z 252.493,A -85,B 0,C 180,E1 -6191.597,E2 -6191.597} C_VEL
LIN {X 0,Y 496.206,Z 267.566,A -85,B 0,C 180,E1 -6193.949,E2 -6193.949} C_VEL
LIN {X 0,Y 498.477,Z 283.976,A -85,B 0,C 180,E1 -6194.268,E2 -6194.268} C_VEL
LIN {X 0,Y 497.966,Z 376.08,A -85,B 0,C 180,E1 -6195.623,E2 -6195.623} C_VEL
LIN {X 0,Y 497.643,Z 389.392,A -85,B 0,C 180,E1 -6195.978,E2 -6195.978} C_VEL
LIN {X 0,Y 497.231,Z 402.714,A -85,B 0,C 180,E1 -6196.513,E2 -6196.513} C_VEL
LIN {X 0,Y 496.904,Z 413.944,A -85,B 0,C 180,E1 -6197.131,E2 -6197.131} C_VEL
LIN {X 0,Y 496.473,Z 425.54,A -85,B 0,C 180,E1 -6197.948,E2 -6197.948} C_VEL
LIN {X 0,Y 496.122,Z 436.023,A -85,B 0,C 180,E1 -6198.871,E2 -6198.871} C_VEL
LIN {X 0,Y 495.809,Z 444.599,A -85,B 0,C 180,E1 -6199.794,E2 -6199.794} C_VEL
LIN {X 0,Y 495.539,Z 452.517,A -85,B 0,C 180,E1 -6200.818,E2 -6200.818} C_VEL
LIN {X 0,Y 495.322,Z 460.256,A -85,B 0,C 180,E1 -6202.048,E2 -6202.048} C_VEL
LIN {X 0,Y 495.165,Z 467.397,A -85,B 0,C 180,E1 -6203.479,E2 -6203.479} C_VEL
LIN {X 0,Y 495.101,Z 472.152,A -85,B 0,C 180,E1 -6204.705,E2 -6204.705} C_VEL
LIN {X 0,Y 495.035,Z 475.785,A -85,B 0,C 180,E1 -6205.928,E2 -6205.928} C_VEL
LIN {X 0,Y 495.042,Z 477.662,A -85,B 0,C 180,E1 -6206.743,E2 -6206.743} C_VEL
LIN {X 0,Y 495.025,Z 479.07,A -85,B 0,C 180,E1 -6207.558,E2 -6207.558} C_VEL
LIN {X 0,Y 494.916,Z 480.686,A -85,B 0,C 180,E1 -6209.185,E2 -6209.185} C_VEL
LIN {X 0,Y 494.909,Z 480.908,A -85,B 0,C 180,E1 -6209.999,E2 -6209.999} C_VEL
LIN {X 0,Y 494.963,Z 480.09,A -85,B 0,C 180,E1 -6211.626,E2 -6211.626} C_VEL
LIN {X 0,Y 495.024,Z 479.096,A -85,B 0,C 180,E1 -6212.439,E2 -6212.439} C_VEL
LIN {X 0,Y 495.041,Z 477.697,A -85,B 0,C 180,E1 -6213.254,E2 -6213.254} C_VEL
LIN {X 0,Y 495.007,Z 474.749,A -85,B 0,C 180,E1 -6214.477,E2 -6214.477} C_VEL
LIN {X 0,Y 495.114,Z 470.764,A -85,B 0,C 180,E1 -6215.701,E2 -6215.701} C_VEL
LIN {X 0,Y 495.202,Z 464.628,A -85,B 0,C 180,E1 -6217.131,E2 -6217.131} C_VEL
LIN {X 0,Y 495.412,Z 457.928,A -85,B 0,C 180,E1 -6218.359,E2 -6218.359} C_VEL
LIN {X 0,Y 495.656,Z 449.612,A -85,B 0,C 180,E1 -6219.588,E2 -6219.588} C_VEL
LIN {X 0,Y 495.947,Z 441.083,A -85,B 0,C 180,E1 -6220.613,E2 -6220.613} C_VEL
LIN {X 0,Y 496.369,Z 430.549,A -85,B 0,C 180,E1 -6221.638,E2 -6221.638} C_VEL
LIN {X 0,Y 496.738,Z 418.688,A -85,B 0,C 180,E1 -6222.561,E2 -6222.561} C_VEL
LIN {X 0,Y 497.12,Z 406.746,A -85,B 0,C 180,E1 -6223.279,E2 -6223.279} C_VEL
LIN {X 0,Y 497.473,Z 394.323,A -85,B 0,C 180,E1 -6223.841,E2 -6223.841} C_VEL
LIN {X 0,Y 497.802,Z 381.533,A -85,B 0,C 180,E1 -6224.249,E2 -6224.249} C_VEL
LIN {X 0,Y 498.051,Z 368.015,A -85,B 0,C 180,E1 -6224.503,E2 -6224.503} C_VEL
LIN {X 0,Y 498.448,Z 282.971,A -85,B 0,C 180,E1 -6225.738,E2 -6225.738} C_VEL
LIN {X 0,Y 496.229,Z 267.738,A -85,B 0,C 180,E1 -6226.034,E2 -6226.034} C_VEL
LIN {X 0,Y 496.733,Z 248.864,A -85,B 0,C 180,E1 -6228.987,E2 -6228.987} C_VEL
LIN {X 0,Y 497.3,Z 229.879,A -85,B 0,C 180,E1 -6231.99,E2 -6231.99} C_VEL
LIN {X 0,Y 497.658,Z 217.649,A -85,B 0,C 180,E1 -6233.95,E2 -6233.95} C_VEL
LIN {X 0,Y 495.833,Z 207.724,A -85,B 0,C 180,E1 -6235.667,E2 -6235.667} C_VEL
LIN {X 0,Y 495.758,Z 207.731,A -85,B 0,C 180,E1 -6238.811,E2 -6238.811} C_VEL
LIN {X 0,Y 495.739,Z 207.732,A -85,B 0,C 180,E1 -6241.722,E2 -6241.722} C_VEL
LIN {X 0,Y 495.757,Z 207.727,A -85,B 0,C 180,E1 -6244.691,E2 -6244.691} C_VEL
LIN {X 0,Y 495.709,Z 207.736,A -85,B 0,C 180,E1 -6247.558,E2 -6247.558} C_VEL
LIN {X 0,Y 495.741,Z 207.729,A -85,B 0,C 180,E1 -6250.696,E2 -6250.696} C_VEL
LIN {X 0,Y 495.705,Z 207.74,A -85,B 0,C 180,E1 -6253.997,E2 -6253.997} C_VEL
LIN {X 0,Y 495.732,Z 207.73,A -85,B 0,C 180,E1 -6257.117,E2 -6257.117} C_VEL
LIN {X 0,Y 495.76,Z 207.727,A -85,B 0,C 180,E1 -6260.362,E2 -6260.362} C_VEL
LIN {X 0,Y 495.696,Z 207.739,A -85,B 0,C 180,E1 -6263.453,E2 -6263.453} C_VEL
LIN {X 0,Y 495.721,Z 207.731,A -85,B 0,C 180,E1 -6266.432,E2 -6266.432} C_VEL
LIN {X 0,Y 495.715,Z 207.736,A -85,B 0,C 180,E1 -6269.31,E2 -6269.31} C_VEL
LIN {X 0,Y 495.739,Z 207.73,A -85,B 0,C 180,E1 -6272.106,E2 -6272.106} C_VEL
LIN {X 0,Y 495.747,Z 207.729,A -85,B 0,C 180,E1 -6274.83,E2 -6274.83} C_VEL
LIN {X 0,Y 495.736,Z 207.737,A -85,B 0,C 180,E1 -6277.494,E2 -6277.494} C_VEL
LIN {X 0,Y 495.728,Z 207.731,A -85,B 0,C 180,E1 -6280.108,E2 -6280.108} C_VEL
LIN {X 0,Y 495.745,Z 207.729,A -85,B 0,C 180,E1 -6282.68,E2 -6282.68} C_VEL
LIN {X 0,Y 495.743,Z 207.735,A -85,B 0,C 180,E1 -6285.215,E2 -6285.215} C_VEL
LIN {X 0,Y 495.826,Z 207.718,A -85,B 0,C 180,E1 -6288.554,E2 -6288.554} C_VEL
LIN {X 0,Y 495.832,Z 207.718,A -85,B 0,C 180,E1 -6291.851,E2 -6291.851} C_VEL
LIN {X 0,Y 495.865,Z 207.713,A -85,B 0,C 180,E1 -6294.306,E2 -6294.306} C_VEL
LIN {X 0,Y 495.937,Z 207.707,A -85,B 0,C 180,E1 -6297.563,E2 -6297.563} C_VEL
LIN {X 0,Y 495.937,Z 207.704,A -85,B 0,C 180,E1 -6300,E2 -6300} C_VEL
LIN {X 0,Y 495.936,Z 207.706,A -85,B 0,C 180,E1 -6302.436,E2 -6302.436} C_VEL
LIN {X 0,Y 495.841,Z 207.717,A -85,B 0,C 180,E1 -6305.694,E2 -6305.694} C_VEL
LIN {X 0,Y 495.818,Z 207.719,A -85,B 0,C 180,E1 -6308.149,E2 -6308.149} C_VEL
LIN {X 0,Y 495.819,Z 207.72,A -85,B 0,C 180,E1 -6311.446,E2 -6311.446} C_VEL
LIN {X 0,Y 495.735,Z 207.738,A -85,B 0,C 180,E1 -6314.784,E2 -6314.784} C_VEL
LIN {X 0,Y 495.742,Z 207.73,A -85,B 0,C 180,E1 -6317.32,E2 -6317.32} C_VEL
LIN {X 0,Y 495.72,Z 207.731,A -85,B 0,C 180,E1 -6319.892,E2 -6319.892} C_VEL
LIN {X 0,Y 495.715,Z 207.738,A -85,B 0,C 180,E1 -6322.864,E2 -6322.864} C_VEL
LIN {X 0,Y 495.743,Z 207.73,A -85,B 0,C 180,E1 -6326.07,E2 -6326.07} C_VEL
LIN {X 0,Y 495.726,Z 207.736,A -85,B 0,C 180,E1 -6328.817,E2 -6328.817} C_VEL
LIN {X 0,Y 495.713,Z 207.732,A -85,B 0,C 180,E1 -6331.728,E2 -6331.728} C_VEL
LIN {X 0,Y 495.733,Z 207.735,A -85,B 0,C 180,E1 -6334.698,E2 -6334.698} C_VEL
LIN {X 0,Y 495.691,Z 207.735,A -85,B 0,C 180,E1 -6337.565,E2 -6337.565} C_VEL
LIN {X 0,Y 495.73,Z 207.734,A -85,B 0,C 180,E1 -6340.703,E2 -6340.703} C_VEL
LIN {X 0,Y 495.694,Z 207.738,A -85,B 0,C 180,E1 -6344.005,E2 -6344.005} C_VEL
LIN {X 0,Y 495.694,Z 207.734,A -85,B 0,C 180,E1 -6347.12,E2 -6347.12} C_VEL
LIN {X 0,Y 495.73,Z 207.735,A -85,B 0,C 180,E1 -6349.957,E2 -6349.957} C_VEL
LIN {X 0,Y 495.704,Z 207.736,A -85,B 0,C 180,E1 -6352.557,E2 -6352.557} C_VEL
LIN {X 0,Y 495.76,Z 207.727,A -85,B 0,C 180,E1 -6355.461,E2 -6355.461} C_VEL
LIN {X 0,Y 495.735,Z 207.734,A -85,B 0,C 180,E1 -6358.367,E2 -6358.367} C_VEL
LIN {X 0,Y 495.734,Z 207.73,A -85,B 0,C 180,E1 -6360.79,E2 -6360.79} C_VEL
LIN {X 0,Y 495.079,Z 207.814,A -85,B 0,C 180,E1 -6361.469,E2 -6361.469} C_VEL
LIN {X 0,Y 492.221,Z 208.169,A -85,B 0,C 180,E1 -6362.572,E2 -6362.572} C_VEL
LIN {X 0,Y 489.807,Z 208.47,A -85,B 0,C 180,E1 -6363.46,E2 -6363.46} C_VEL
LIN {X 0,Y 488.785,Z 208.601,A -85,B 0,C 180,E1 -6364.147,E2 -6364.147} C_VEL
LIN {X 0,Y 488.71,Z 208.606,A -85,B 0,C 180,E1 -6364.379,E2 -6364.379} C_VEL
LIN {X 0,Y 488.709,Z 208.605,A -85,B 0,C 180,E1 -6367.156,E2 -6367.156} C_VEL
LIN {X 0,Y 488.712,Z 208.612,A -85,B 0,C 180,E1 -6369.813,E2 -6369.813} C_VEL
LIN {X 0,Y 488.698,Z 208.607,A -85,B 0,C 180,E1 -6372.425,E2 -6372.425} C_VEL
LIN {X 0,Y 488.749,Z 208.6,A -85,B 0,C 180,E1 -6375.002,E2 -6375.002} C_VEL
LIN {X 0,Y 488.8,Z 208.594,A -85,B 0,C 180,E1 -6378.39,E2 -6378.39} C_VEL
LIN {X 0,Y 488.782,Z 208.604,A -85,B 0,C 180,E1 -6381.735,E2 -6381.735} C_VEL
LIN {X 0,Y 488.836,Z 208.595,A -85,B 0,C 180,E1 -6384.226,E2 -6384.226} C_VEL
LIN {X 0,Y 488.822,Z 208.718,A -85,B 0,C 180,E1 -6385.518,E2 -6385.518} C_VEL
LIN {X 0,Y 489.469,Z 214.553,A -85,B 0,C 180,E1 -6386.709,E2 -6386.709} C_VEL
LIN {X 0,Y 489.347,Z 225.174,A -85,B 0,C 180,E1 -6388.809,E2 -6388.809} C_VEL
LIN {X 0,Y 491.731,Z 237.251,A -85,B 0,C 180,E1 -6389.074,E2 -6389.074} C_VEL
LIN {X 0,Y 491.133,Z 332.124,A -85,B 0,C 180,E1 -6390.488,E2 -6390.488} C_VEL
LIN {X 0,Y 490.921,Z 345.21,A -85,B 0,C 180,E1 -6390.847,E2 -6390.847} C_VEL
LIN {X 0,Y 490.661,Z 358.33,A -85,B 0,C 180,E1 -6391.386,E2 -6391.386} C_VEL
LIN {X 0,Y 490.283,Z 370.208,A -85,B 0,C 180,E1 -6392.055,E2 -6392.055} C_VEL
LIN {X 0,Y 489.807,Z 381.585,A -85,B 0,C 180,E1 -6392.88,E2 -6392.88} C_VEL
LIN {X 0,Y 489.422,Z 391.823,A -85,B 0,C 180,E1 -6393.809,E2 -6393.809} C_VEL
LIN {X 0,Y 489.086,Z 400.217,A -85,B 0,C 180,E1 -6394.74,E2 -6394.74} C_VEL
LIN {X 0,Y 488.713,Z 409.332,A -85,B 0,C 180,E1 -6395.985,E2 -6395.985} C_VEL
LIN {X 0,Y 488.517,Z 416.556,A -85,B 0,C 180,E1 -6397.212,E2 -6397.212} C_VEL
LIN {X 0,Y 488.329,Z 421.668,A -85,B 0,C 180,E1 -6398.275,E2 -6398.275} C_VEL
LIN {X 0,Y 488.136,Z 426.536,A -85,B 0,C 180,E1 -6399.531,E2 -6399.531} C_VEL
LIN {X 0,Y 488.032,Z 430.279,A -85,B 0,C 180,E1 -6400.79,E2 -6400.79} C_VEL
LIN {X 0,Y 487.998,Z 432.303,A -85,B 0,C 180,E1 -6401.675,E2 -6401.675} C_VEL
LIN {X 0,Y 487.92,Z 433.703,A -85,B 0,C 180,E1 -6402.478,E2 -6402.478} C_VEL
LIN {X 0,Y 487.866,Z 434.746,A -85,B 0,C 180,E1 -6403.326,E2 -6403.326} C_VEL
LIN {X 0,Y 487.867,Z 435.389,A -85,B 0,C 180,E1 -6404.176,E2 -6404.176} C_VEL
LIN {X 0,Y 487.881,Z 435.617,A -85,B 0,C 180,E1 -6405.173,E2 -6405.173} C_VEL
LIN {X 0,Y 487.835,Z 434.79,A -85,B 0,C 180,E1 -6406.746,E2 -6406.746} C_VEL
LIN {X 0,Y 487.935,Z 432.966,A -85,B 0,C 180,E1 -6408.079,E2 -6408.079} C_VEL
LIN {X 0,Y 488.076,Z 429.072,A -85,B 0,C 180,E1 -6409.778,E2 -6409.778} C_VEL
LIN {X 0,Y 488.211,Z 424.724,A -85,B 0,C 180,E1 -6411.093,E2 -6411.093} C_VEL
LIN {X 0,Y 488.401,Z 419.041,A -85,B 0,C 180,E1 -6412.415,E2 -6412.415} C_VEL
LIN {X 0,Y 488.683,Z 411.81,A -85,B 0,C 180,E1 -6413.745,E2 -6413.745} C_VEL
LIN {X 0,Y 488.982,Z 404.08,A -85,B 0,C 180,E1 -6414.885,E2 -6414.885} C_VEL
LIN {X 0,Y 489.355,Z 394.974,A -85,B 0,C 180,E1 -6415.978,E2 -6415.978} C_VEL
LIN {X 0,Y 489.738,Z 384.856,A -85,B 0,C 180,E1 -6416.966,E2 -6416.966} C_VEL
LIN {X 0,Y 490.17,Z 374.616,A -85,B 0,C 180,E1 -6417.773,E2 -6417.773} C_VEL
LIN {X 0,Y 490.577,Z 362.843,A -85,B 0,C 180,E1 -6418.504,E2 -6418.504} C_VEL
LIN {X 0,Y 490.876,Z 350.426,A -85,B 0,C 180,E1 -6419.086,E2 -6419.086} C_VEL
LIN {X 0,Y 491.094,Z 338.09,A -85,B 0,C 180,E1 -6419.496,E2 -6419.496} C_VEL
LIN {X 0,Y 491.238,Z 324.587,A -85,B 0,C 180,E1 -6419.766,E2 -6419.766} C_VEL
LIN {X 0,Y 491.787,Z 237.039,A -85,B 0,C 180,E1 -6421.061,E2 -6421.061} C_VEL
LIN {X 0,Y 489.361,Z 225.24,A -85,B 0,C 180,E1 -6421.336,E2 -6421.336} C_VEL
LIN {X 0,Y 489.525,Z 212.603,A -85,B 0,C 180,E1 -6423.788,E2 -6423.788} C_VEL
LIN {X 0,Y 488.767,Z 208.605,A -85,B 0,C 180,E1 -6424.607,E2 -6424.607} C_VEL
LIN {X 0,Y 488.672,Z 208.617,A -85,B 0,C 180,E1 -6428.198,E2 -6428.198} C_VEL
LIN {X 0,Y 488.738,Z 208.61,A -85,B 0,C 180,E1 -6430.348,E2 -6430.348} C_VEL
LIN {X 0,Y 488.702,Z 208.61,A -85,B 0,C 180,E1 -6433.65,E2 -6433.65} C_VEL
LIN {X 0,Y 488.7,Z 208.614,A -85,B 0,C 180,E1 -6436.347,E2 -6436.347} C_VEL
LIN {X 0,Y 488.715,Z 208.608,A -85,B 0,C 180,E1 -6439.675,E2 -6439.675} C_VEL
LIN {X 0,Y 488.66,Z 208.616,A -85,B 0,C 180,E1 -6442.276,E2 -6442.276} C_VEL
LIN {X 0,Y 488.707,Z 208.604,A -85,B 0,C 180,E1 -6445.05,E2 -6445.05} C_VEL
LIN {X 0,Y 488.683,Z 208.612,A -85,B 0,C 180,E1 -6448.044,E2 -6448.044} C_VEL
LIN {X 0,Y 488.709,Z 208.603,A -85,B 0,C 180,E1 -6450.729,E2 -6450.729} C_VEL
LIN {X 0,Y 488.732,Z 208.605,A -85,B 0,C 180,E1 -6453.527,E2 -6453.527} C_VEL
LIN {X 0,Y 488.684,Z 208.61,A -85,B 0,C 180,E1 -6456.254,E2 -6456.254} C_VEL
LIN {X 0,Y 488.72,Z 208.602,A -85,B 0,C 180,E1 -6459.174,E2 -6459.174} C_VEL
LIN {X 0,Y 488.711,Z 208.602,A -85,B 0,C 180,E1 -6462.423,E2 -6462.423} C_VEL
LIN {X 0,Y 488.734,Z 208.603,A -85,B 0,C 180,E1 -6464.999,E2 -6464.999} C_VEL
LIN {X 0,Y 488.776,Z 208.596,A -85,B 0,C 180,E1 -6468.387,E2 -6468.387} C_VEL
LIN {X 0,Y 488.789,Z 208.596,A -85,B 0,C 180,E1 -6471.733,E2 -6471.733} C_VEL
LIN {X 0,Y 488.835,Z 208.589,A -85,B 0,C 180,E1 -6474.224,E2 -6474.224} C_VEL
LIN {X 0,Y 488.927,Z 208.581,A -85,B 0,C 180,E1 -6477.529,E2 -6477.529} C_VEL
LIN {X 0,Y 488.931,Z 208.574,A -85,B 0,C 180,E1 -6480,E2 -6480} C_VEL
LIN {X 0,Y 488.926,Z 208.575,A -85,B 0,C 180,E1 -6482.472,E2 -6482.472} C_VEL
LIN {X 0,Y 488.813,Z 208.588,A -85,B 0,C 180,E1 -6485.777,E2 -6485.777} C_VEL
LIN {X 0,Y 488.754,Z 208.598,A -85,B 0,C 180,E1 -6488.268,E2 -6488.268} C_VEL
LIN {X 0,Y 488.803,Z 208.593,A -85,B 0,C 180,E1 -6491.613,E2 -6491.613} C_VEL
LIN {X 0,Y 488.73,Z 208.605,A -85,B 0,C 180,E1 -6495.002,E2 -6495.002} C_VEL
LIN {X 0,Y 488.718,Z 208.606,A -85,B 0,C 180,E1 -6498.444,E2 -6498.444} C_VEL
LIN {X 0,Y 488.679,Z 208.613,A -85,B 0,C 180,E1 -6501.072,E2 -6501.072} C_VEL
LIN {X 0,Y 488.641,Z 208.611,A -85,B 0,C 180,E1 -6503.748,E2 -6503.748} C_VEL
LIN {X 0,Y 488.699,Z 208.609,A -85,B 0,C 180,E1 -6506.929,E2 -6506.929} C_VEL
LIN {X 0,Y 488.699,Z 208.61,A -85,B 0,C 180,E1 -6510.221,E2 -6510.221} C_VEL
LIN {X 0,Y 488.689,Z 208.607,A -85,B 0,C 180,E1 -6513.481,E2 -6513.481} C_VEL
LIN {X 0,Y 488.653,Z 208.619,A -85,B 0,C 180,E1 -6516.355,E2 -6516.355} C_VEL
LIN {X 0,Y 488.678,Z 208.61,A -85,B 0,C 180,E1 -6519.257,E2 -6519.257} C_VEL
LIN {X 0,Y 488.683,Z 208.604,A -85,B 0,C 180,E1 -6521.6,E2 -6521.6} C_VEL
LIN {X 0,Y 488.688,Z 208.609,A -85,B 0,C 180,E1 -6524.805,E2 -6524.805} C_VEL
LIN {X 0,Y 488.677,Z 208.61,A -85,B 0,C 180,E1 -6527.476,E2 -6527.476} C_VEL
LIN {X 0,Y 488.684,Z 208.61,A -85,B 0,C 180,E1 -6530.747,E2 -6530.747} C_VEL
LIN {X 0,Y 488.671,Z 208.613,A -85,B 0,C 180,E1 -6533.87,E2 -6533.87} C_VEL
LIN {X 0,Y 488.733,Z 208.604,A -85,B 0,C 180,E1 -6536.879,E2 -6536.879} C_VEL
LIN {X 0,Y 488.72,Z 208.609,A -85,B 0,C 180,E1 -6539.782,E2 -6539.782} C_VEL
LIN {X 0,Y 488.723,Z 208.608,A -85,B 0,C 180,E1 -6543.073,E2 -6543.073} C_VEL
LIN {X 0,Y 488.736,Z 208.614,A -85,B 0,C 180,E1 -6544.102,E2 -6544.102} C_VEL
LIN {X 0,Y 490.698,Z 218.805,A -85,B 0,C 180,E1 -6545.91,E2 -6545.91} C_VEL
LIN {X 0,Y 490.405,Z 229.614,A -85,B 0,C 180,E1 -6547.681,E2 -6547.681} C_VEL
LIN {X 0,Y 489.798,Z 248.498,A -85,B 0,C 180,E1 -6550.73,E2 -6550.73} C_VEL
LIN {X 0,Y 489.246,Z 267.401,A -85,B 0,C 180,E1 -6553.706,E2 -6553.706} C_VEL
LIN {X 0,Y 491.68,Z 284.287,A -85,B 0,C 180,E1 -6554.045,E2 -6554.045} C_VEL
LIN {X 0,Y 491.108,Z 375.983,A -85,B 0,C 180,E1 -6555.417,E2 -6555.417} C_VEL
LIN {X 0,Y 490.775,Z 389.192,A -85,B 0,C 180,E1 -6555.778,E2 -6555.778} C_VEL
LIN {X 0,Y 490.306,Z 402.453,A -85,B 0,C 180,E1 -6556.319,E2 -6556.319} C_VEL
LIN {X 0,Y 489.947,Z 413.939,A -85,B 0,C 180,E1 -6556.964,E2 -6556.964} C_VEL
LIN {X 0,Y 489.515,Z 425.247,A -85,B 0,C 180,E1 -6557.774,E2 -6557.774} C_VEL
LIN {X 0,Y 489.129,Z 435.724,A -85,B 0,C 180,E1 -6558.71,E2 -6558.71} C_VEL
LIN {X 0,Y 488.784,Z 444.294,A -85,B 0,C 180,E1 -6559.645,E2 -6559.645} C_VEL
LIN {X 0,Y 488.478,Z 452.206,A -85,B 0,C 180,E1 -6560.685,E2 -6560.685} C_VEL
LIN {X 0,Y 488.251,Z 459.942,A -85,B 0,C 180,E1 -6561.932,E2 -6561.932} C_VEL
LIN {X 0,Y 488.074,Z 467.076,A -85,B 0,C 180,E1 -6563.384,E2 -6563.384} C_VEL
LIN {X 0,Y 488.011,Z 471.828,A -85,B 0,C 180,E1 -6564.628,E2 -6564.628} C_VEL
LIN {X 0,Y 487.931,Z 475.459,A -85,B 0,C 180,E1 -6565.869,E2 -6565.869} C_VEL
LIN {X 0,Y 487.965,Z 477.336,A -85,B 0,C 180,E1 -6566.696,E2 -6566.696} C_VEL
LIN {X 0,Y 487.933,Z 478.743,A -85,B 0,C 180,E1 -6567.522,E2 -6567.522} C_VEL
LIN {X 0,Y 487.892,Z 479.747,A -85,B 0,C 180,E1 -6568.348,E2 -6568.348} C_VEL
LIN {X 0,Y 487.829,Z 480.581,A -85,B 0,C 180,E1 -6569.999,E2 -6569.999} C_VEL
LIN {X 0,Y 487.892,Z 479.764,A -85,B 0,C 180,E1 -6571.649,E2 -6571.649} C_VEL
LIN {X 0,Y 487.932,Z 478.768,A -85,B 0,C 180,E1 -6572.475,E2 -6572.475} C_VEL
LIN {X 0,Y 487.964,Z 477.369,A -85,B 0,C 180,E1 -6573.301,E2 -6573.301} C_VEL
LIN {X 0,Y 487.919,Z 474.418,A -85,B 0,C 180,E1 -6574.542,E2 -6574.542} C_VEL
LIN {X 0,Y 488.01,Z 470.427,A -85,B 0,C 180,E1 -6575.784,E2 -6575.784} C_VEL
LIN {X 0,Y 488.129,Z 464.284,A -85,B 0,C 180,E1 -6577.235,E2 -6577.235} C_VEL
LIN {X 0,Y 488.343,Z 457.574,A -85,B 0,C 180,E1 -6578.481,E2 -6578.481} C_VEL
LIN {X 0,Y 488.59,Z 449.247,A -85,B 0,C 180,E1 -6579.728,E2 -6579.728} C_VEL
LIN {X 0,Y 488.923,Z 440.709,A -85,B 0,C 180,E1 -6580.768,E2 -6580.768} C_VEL
LIN {X 0,Y 489.381,Z 430.163,A -85,B 0,C 180,E1 -6581.806,E2 -6581.806} C_VEL
LIN {X 0,Y 489.769,Z 418.584,A -85,B 0,C 180,E1 -6582.722,E2 -6582.722} C_VEL
LIN {X 0,Y 490.191,Z 406.318,A -85,B 0,C 180,E1 -6583.47,E2 -6583.47} C_VEL
LIN {X 0,Y 490.588,Z 393.865,A -85,B 0,C 180,E1 -6584.04,E2 -6584.04} C_VEL
LIN {X 0,Y 490.933,Z 381.001,A -85,B 0,C 180,E1 -6584.453,E2 -6584.453} C_VEL
LIN {X 0,Y 491.172,Z 367.322,A -85,B 0,C 180,E1 -6584.71,E2 -6584.71} C_VEL
LIN {X 0,Y 491.447,Z 282.746,A -85,B 0,C 180,E1 -6585.96,E2 -6585.96} C_VEL
LIN {X 0,Y 489.22,Z 267.38,A -85,B 0,C 180,E1 -6586.265,E2 -6586.265} C_VEL
LIN {X 0,Y 489.773,Z 248.468,A -85,B 0,C 180,E1 -6589.268,E2 -6589.268} C_VEL
LIN {X 0,Y 490.399,Z 229.473,A -85,B 0,C 180,E1 -6592.316,E2 -6592.316} C_VEL
LIN {X 0,Y 490.663,Z 218.554,A -85,B 0,C 180,E1 -6594.089,E2 -6594.089} C_VEL
LIN {X 0,Y 488.781,Z 208.603,A -85,B 0,C 180,E1 -6595.835,E2 -6595.835} C_VEL
LIN {X 0,Y 488.718,Z 208.609,A -85,B 0,C 180,E1 -6598.692,E2 -6598.692} C_VEL
LIN {X 0,Y 488.676,Z 208.609,A -85,B 0,C 180,E1 -6601.176,E2 -6601.176} C_VEL
LIN {X 0,Y 488.717,Z 208.611,A -85,B 0,C 180,E1 -6604.109,E2 -6604.109} C_VEL
LIN {X 0,Y 488.66,Z 208.611,A -85,B 0,C 180,E1 -6607.155,E2 -6607.155} C_VEL
LIN {X 0,Y 488.694,Z 208.609,A -85,B 0,C 180,E1 -6610.341,E2 -6610.341} C_VEL
LIN {X 0,Y 488.658,Z 208.616,A -85,B 0,C 180,E1 -6613.651,E2 -6613.651} C_VEL
LIN {X 0,Y 488.686,Z 208.609,A -85,B 0,C 180,E1 -6616.345,E2 -6616.345} C_VEL
LIN {X 0,Y 488.737,Z 208.608,A -85,B 0,C 180,E1 -6619.677,E2 -6619.677} C_VEL
LIN {X 0,Y 488.646,Z 208.612,A -85,B 0,C 180,E1 -6622.838,E2 -6622.838} C_VEL
LIN {X 0,Y 488.695,Z 208.611,A -85,B 0,C 180,E1 -6625.884,E2 -6625.884} C_VEL
LIN {X 0,Y 488.654,Z 208.612,A -85,B 0,C 180,E1 -6628.817,E2 -6628.817} C_VEL
LIN {X 0,Y 488.704,Z 208.612,A -85,B 0,C 180,E1 -6631.668,E2 -6631.668} C_VEL
LIN {X 0,Y 488.707,Z 208.605,A -85,B 0,C 180,E1 -6634.442,E2 -6634.442} C_VEL
LIN {X 0,Y 488.703,Z 208.609,A -85,B 0,C 180,E1 -6637.152,E2 -6637.152} C_VEL
LIN {X 0,Y 488.68,Z 208.611,A -85,B 0,C 180,E1 -6639.808,E2 -6639.808} C_VEL
LIN {X 0,Y 488.689,Z 208.607,A -85,B 0,C 180,E1 -6642.421,E2 -6642.421} C_VEL
LIN {X 0,Y 488.713,Z 208.608,A -85,B 0,C 180,E1 -6644.998,E2 -6644.998} C_VEL
LIN {X 0,Y 488.783,Z 208.595,A -85,B 0,C 180,E1 -6648.387,E2 -6648.387} C_VEL
LIN {X 0,Y 488.794,Z 208.596,A -85,B 0,C 180,E1 -6651.733,E2 -6651.733} C_VEL
LIN {X 0,Y 488.822,Z 208.59,A -85,B 0,C 180,E1 -6654.224,E2 -6654.224} C_VEL
LIN {X 0,Y 488.905,Z 208.583,A -85,B 0,C 180,E1 -6657.528,E2 -6657.528} C_VEL
LIN {X 0,Y 488.909,Z 208.58,A -85,B 0,C 180,E1 -6660,E2 -6660} C_VEL
LIN {X 0,Y 488.904,Z 208.582,A -85,B 0,C 180,E1 -6662.471,E2 -6662.471} C_VEL
LIN {X 0,Y 488.798,Z 208.594,A -85,B 0,C 180,E1 -6665.776,E2 -6665.776} C_VEL
LIN {X 0,Y 488.763,Z 208.599,A -85,B 0,C 180,E1 -6668.267,E2 -6668.267} C_VEL
LIN {X 0,Y 488.779,Z 208.596,A -85,B 0,C 180,E1 -6671.613,E2 -6671.613} C_VEL
LIN {X 0,Y 488.707,Z 208.611,A -85,B 0,C 180,E1 -6675.002,E2 -6675.002} C_VEL
LIN {X 0,Y 488.708,Z 208.608,A -85,B 0,C 180,E1 -6678.374,E2 -6678.374} C_VEL
LIN {X 0,Y 488.661,Z 208.614,A -85,B 0,C 180,E1 -6681.073,E2 -6681.073} C_VEL
LIN {X 0,Y 488.65,Z 208.612,A -85,B 0,C 180,E1 -6683.747,E2 -6683.747} C_VEL
LIN {X 0,Y 488.745,Z 208.604,A -85,B 0,C 180,E1 -6686.946,E2 -6686.946} C_VEL
LIN {X 0,Y 488.664,Z 208.616,A -85,B 0,C 180,E1 -6690.365,E2 -6690.365} C_VEL
LIN {X 0,Y 488.693,Z 208.606,A -85,B 0,C 180,E1 -6693.487,E2 -6693.487} C_VEL
LIN {X 0,Y 488.648,Z 208.619,A -85,B 0,C 180,E1 -6696.359,E2 -6696.359} C_VEL
LIN {X 0,Y 488.662,Z 208.61,A -85,B 0,C 180,E1 -6699.258,E2 -6699.258} C_VEL
LIN {X 0,Y 488.672,Z 208.609,A -85,B 0,C 180,E1 -6701.603,E2 -6701.603} C_VEL
LIN {X 0,Y 488.668,Z 208.612,A -85,B 0,C 180,E1 -6704.806,E2 -6704.806} C_VEL
LIN {X 0,Y 488.661,Z 208.611,A -85,B 0,C 180,E1 -6707.478,E2 -6707.478} C_VEL
LIN {X 0,Y 488.705,Z 208.607,A -85,B 0,C 180,E1 -6709.68,E2 -6709.68} C_VEL
LIN {X 0,Y 488.656,Z 208.612,A -85,B 0,C 180,E1 -6712.845,E2 -6712.845} C_VEL
LIN {X 0,Y 488.711,Z 208.609,A -85,B 0,C 180,E1 -6715.891,E2 -6715.891} C_VEL
LIN {X 0,Y 488.672,Z 208.61,A -85,B 0,C 180,E1 -6718.824,E2 -6718.824} C_VEL
LIN {X 0,Y 488.726,Z 208.606,A -85,B 0,C 180,E1 -6721.675,E2 -6721.675} C_VEL
LIN {X 0,Y 488.71,Z 208.606,A -85,B 0,C 180,E1 -6724.379,E2 -6724.379} C_VEL
LIN {X 0,Y 488.061,Z 208.691,A -85,B 0,C 180,E1 -6725.067,E2 -6725.067} C_VEL
LIN {X 0,Y 485.197,Z 209.052,A -85,B 0,C 180,E1 -6726.184,E2 -6726.184} C_VEL
LIN {X 0,Y 482.76,Z 209.353,A -85,B 0,C 180,E1 -6727.084,E2 -6727.084} C_VEL
LIN {X 0,Y 481.709,Z 209.483,A -85,B 0,C 180,E1 -6727.78,E2 -6727.78} C_VEL
LIN {X 0,Y 481.621,Z 209.49,A -85,B 0,C 180,E1 -6728.016,E2 -6728.016} C_VEL
LIN {X 0,Y 481.691,Z 209.481,A -85,B 0,C 180,E1 -6730.396,E2 -6730.396} C_VEL
LIN {X 0,Y 481.663,Z 209.482,A -85,B 0,C 180,E1 -6733.036,E2 -6733.036} C_VEL
LIN {X 0,Y 481.675,Z 209.487,A -85,B 0,C 180,E1 -6735.641,E2 -6735.641} C_VEL
LIN {X 0,Y 481.745,Z 209.474,A -85,B 0,C 180,E1 -6738.218,E2 -6738.218} C_VEL
LIN {X 0,Y 481.736,Z 209.481,A -85,B 0,C 180,E1 -6741.613,E2 -6741.613} C_VEL
LIN {X 0,Y 481.794,Z 209.472,A -85,B 0,C 180,E1 -6744.141,E2 -6744.141} C_VEL
LIN {X 0,Y 481.807,Z 209.675,A -85,B 0,C 180,E1 -6745.4,E2 -6745.4} C_VEL
LIN {X 0,Y 482.487,Z 215.802,A -85,B 0,C 180,E1 -6746.662,E2 -6746.662} C_VEL
LIN {X 0,Y 482.376,Z 225.461,A -85,B 0,C 180,E1 -6748.584,E2 -6748.584} C_VEL
LIN {X 0,Y 484.98,Z 239.133,A -85,B 0,C 180,E1 -6748.883,E2 -6748.883} C_VEL
LIN {X 0,Y 484.27,Z 332.274,A -85,B 0,C 180,E1 -6750.287,E2 -6750.287} C_VEL
LIN {X 0,Y 484.064,Z 344.663,A -85,B 0,C 180,E1 -6750.625,E2 -6750.625} C_VEL
LIN {X 0,Y 483.755,Z 357.48,A -85,B 0,C 180,E1 -6751.146,E2 -6751.146} C_VEL
LIN {X 0,Y 483.429,Z 368.86,A -85,B 0,C 180,E1 -6751.772,E2 -6751.772} C_VEL
LIN {X 0,Y 482.903,Z 380.6,A -85,B 0,C 180,E1 -6752.608,E2 -6752.608} C_VEL
LIN {X 0,Y 482.508,Z 391.067,A -85,B 0,C 180,E1 -6753.55,E2 -6753.55} C_VEL
LIN {X 0,Y 482.098,Z 400.537,A -85,B 0,C 180,E1 -6754.6,E2 -6754.6} C_VEL
LIN {X 0,Y 481.694,Z 409.663,A -85,B 0,C 180,E1 -6755.863,E2 -6755.863} C_VEL
LIN {X 0,Y 481.488,Z 416.312,A -85,B 0,C 180,E1 -6756.997,E2 -6756.997} C_VEL
LIN {X 0,Y 481.231,Z 422.917,A -85,B 0,C 180,E1 -6758.398,E2 -6758.398} C_VEL
LIN {X 0,Y 481.056,Z 427.592,A -85,B 0,C 180,E1 -6759.673,E2 -6759.673} C_VEL
LIN {X 0,Y 480.937,Z 431.156,A -85,B 0,C 180,E1 -6760.952,E2 -6760.952} C_VEL
LIN {X 0,Y 480.892,Z 432.96,A -85,B 0,C 180,E1 -6761.807,E2 -6761.807} C_VEL
LIN {X 0,Y 480.816,Z 434.323,A -85,B 0,C 180,E1 -6762.665,E2 -6762.665} C_VEL
LIN {X 0,Y 480.767,Z 435.283,A -85,B 0,C 180,E1 -6763.527,E2 -6763.527} C_VEL
LIN {X 0,Y 480.799,Z 435.833,A -85,B 0,C 180,E1 -6764.389,E2 -6764.389} C_VEL
LIN {X 0,Y 480.787,Z 435.93,A -85,B 0,C 180,E1 -6765.255,E2 -6765.255} C_VEL
LIN {X 0,Y 480.746,Z 435.622,A -85,B 0,C 180,E1 -6766.127,E2 -6766.127} C_VEL
LIN {X 0,Y 480.753,Z 434.907,A -85,B 0,C 180,E1 -6767,E2 -6767} C_VEL
LIN {X 0,Y 480.878,Z 433.168,A -85,B 0,C 180,E1 -6768.201,E2 -6768.201} C_VEL
LIN {X 0,Y 480.976,Z 430.002,A -85,B 0,C 180,E1 -6769.638,E2 -6769.638} C_VEL
LIN {X 0,Y 481.145,Z 425.589,A -85,B 0,C 180,E1 -6771.048,E2 -6771.048} C_VEL
LIN {X 0,Y 481.295,Z 420.418,A -85,B 0,C 180,E1 -6772.312,E2 -6772.312} C_VEL
LIN {X 0,Y 481.606,Z 413.438,A -85,B 0,C 180,E1 -6773.659,E2 -6773.659} C_VEL
LIN {X 0,Y 481.93,Z 406.213,A -85,B 0,C 180,E1 -6774.787,E2 -6774.787} C_VEL
LIN {X 0,Y 482.348,Z 396.358,A -85,B 0,C 180,E1 -6776.035,E2 -6776.035} C_VEL
LIN {X 0,Y 482.74,Z 386.876,A -85,B 0,C 180,E1 -6776.999,E2 -6776.999} C_VEL
LIN {X 0,Y 483.215,Z 376.502,A -85,B 0,C 180,E1 -6777.854,E2 -6777.854} C_VEL
LIN {X 0,Y 483.605,Z 366.189,A -85,B 0,C 180,E1 -6778.538,E2 -6778.538} C_VEL
LIN {X 0,Y 483.964,Z 353.86,A -85,B 0,C 180,E1 -6779.173,E2 -6779.173} C_VEL
LIN {X 0,Y 484.234,Z 340.46,A -85,B 0,C 180,E1 -6779.657,E2 -6779.657} C_VEL
LIN {X 0,Y 484.394,Z 327.747,A -85,B 0,C 180,E1 -6779.945,E2 -6779.945} C_VEL
LIN {X 0,Y 485.068,Z 238.278,A -85,B 0,C 180,E1 -6781.29,E2 -6781.29} C_VEL
LIN {X 0,Y 482.453,Z 225.457,A -85,B 0,C 180,E1 -6781.607,E2 -6781.607} C_VEL
LIN {X 0,Y 482.568,Z 213.834,A -85,B 0,C 180,E1 -6783.888,E2 -6783.888} C_VEL
LIN {X 0,Y 481.7,Z 209.484,A -85,B 0,C 180,E1 -6784.826,E2 -6784.826} C_VEL
LIN {X 0,Y 481.647,Z 209.491,A -85,B 0,C 180,E1 -6788.006,E2 -6788.006} C_VEL
LIN {X 0,Y 481.674,Z 209.485,A -85,B 0,C 180,E1 -6790.649,E2 -6790.649} C_VEL
LIN {X 0,Y 481.67,Z 209.485,A -85,B 0,C 180,E1 -6793.293,E2 -6793.293} C_VEL
LIN {X 0,Y 481.673,Z 209.484,A -85,B 0,C 180,E1 -6796.844,E2 -6796.844} C_VEL
LIN {X 0,Y 481.671,Z 209.487,A -85,B 0,C 180,E1 -6800.059,E2 -6800.059} C_VEL
LIN {X 0,Y 481.608,Z 209.49,A -85,B 0,C 180,E1 -6803.252,E2 -6803.252} C_VEL
LIN {X 0,Y 481.689,Z 209.483,A -85,B 0,C 180,E1 -6806.329,E2 -6806.329} C_VEL
LIN {X 0,Y 481.634,Z 209.487,A -85,B 0,C 180,E1 -6809.415,E2 -6809.415} C_VEL
LIN {X 0,Y 481.676,Z 209.484,A -85,B 0,C 180,E1 -6812.167,E2 -6812.167} C_VEL
LIN {X 0,Y 481.696,Z 209.475,A -85,B 0,C 180,E1 -6814.969,E2 -6814.969} C_VEL
LIN {X 0,Y 481.648,Z 209.49,A -85,B 0,C 180,E1 -6817.705,E2 -6817.705} C_VEL
LIN {X 0,Y 481.68,Z 209.481,A -85,B 0,C 180,E1 -6820.392,E2 -6820.392} C_VEL
LIN {X 0,Y 481.669,Z 209.481,A -85,B 0,C 180,E1 -6823.033,E2 -6823.033} C_VEL
LIN {X 0,Y 481.664,Z 209.489,A -85,B 0,C 180,E1 -6825.638,E2 -6825.638} C_VEL
LIN {X 0,Y 481.721,Z 209.475,A -85,B 0,C 180,E1 -6828.215,E2 -6828.215} C_VEL
LIN {X 0,Y 481.734,Z 209.475,A -85,B 0,C 180,E1 -6831.611,E2 -6831.611} C_VEL
LIN {X 0,Y 481.797,Z 209.466,A -85,B 0,C 180,E1 -6834.14,E2 -6834.14} C_VEL
LIN {X 0,Y 481.894,Z 209.458,A -85,B 0,C 180,E1 -6837.493,E2 -6837.493} C_VEL
LIN {X 0,Y 481.874,Z 209.456,A -85,B 0,C 180,E1 -6840.836,E2 -6840.836} C_VEL
LIN {X 0,Y 481.893,Z 209.451,A -85,B 0,C 180,E1 -6842.508,E2 -6842.508} C_VEL
LIN {X 0,Y 481.772,Z 209.464,A -85,B 0,C 180,E1 -6845.861,E2 -6845.861} C_VEL
LIN {X 0,Y 481.709,Z 209.476,A -85,B 0,C 180,E1 -6848.39,E2 -6848.39} C_VEL
LIN {X 0,Y 481.767,Z 209.468,A -85,B 0,C 180,E1 -6851.785,E2 -6851.785} C_VEL
LIN {X 0,Y 481.695,Z 209.477,A -85,B 0,C 180,E1 -6855.659,E2 -6855.659} C_VEL
LIN {X 0,Y 481.68,Z 209.484,A -85,B 0,C 180,E1 -6858.723,E2 -6858.723} C_VEL
LIN {X 0,Y 481.617,Z 209.489,A -85,B 0,C 180,E1 -6861.396,E2 -6861.396} C_VEL
LIN {X 0,Y 481.62,Z 209.487,A -85,B 0,C 180,E1 -6864.116,E2 -6864.116} C_VEL
LIN {X 0,Y 481.669,Z 209.482,A -85,B 0,C 180,E1 -6867.128,E2 -6867.128} C_VEL
LIN {X 0,Y 481.649,Z 209.485,A -85,B 0,C 180,E1 -6869.743,E2 -6869.743} C_VEL
LIN {X 0,Y 481.631,Z 209.493,A -85,B 0,C 180,E1 -6872.678,E2 -6872.678} C_VEL
LIN {X 0,Y 481.611,Z 209.49,A -85,B 0,C 180,E1 -6875.712,E2 -6875.712} C_VEL
LIN {X 0,Y 481.648,Z 209.488,A -85,B 0,C 180,E1 -6878.862,E2 -6878.862} C_VEL
LIN {X 0,Y 481.633,Z 209.484,A -85,B 0,C 180,E1 -6881.914,E2 -6881.914} C_VEL
LIN {X 0,Y 481.642,Z 209.491,A -85,B 0,C 180,E1 -6884.46,E2 -6884.46} C_VEL
LIN {X 0,Y 481.629,Z 209.491,A -85,B 0,C 180,E1 -6887.84,E2 -6887.84} C_VEL
LIN {X 0,Y 481.657,Z 209.485,A -85,B 0,C 180,E1 -6891.142,E2 -6891.142} C_VEL
LIN {X 0,Y 481.631,Z 209.494,A -85,B 0,C 180,E1 -6894.292,E2 -6894.292} C_VEL
LIN {X 0,Y 481.667,Z 209.486,A -85,B 0,C 180,E1 -6897.327,E2 -6897.327} C_VEL
LIN {X 0,Y 481.67,Z 209.489,A -85,B 0,C 180,E1 -6900.26,E2 -6900.26} C_VEL
LIN {X 0,Y 481.685,Z 209.487,A -85,B 0,C 180,E1 -6903.577,E2 -6903.577} C_VEL
LIN {X 0,Y 481.704,Z 209.621,A -85,B 0,C 180,E1 -6903.899,E2 -6903.899} C_VEL
LIN {X 0,Y 483.747,Z 219.957,A -85,B 0,C 180,E1 -6905.769,E2 -6905.769} C_VEL
LIN {X 0,Y 483.698,Z 226.701,A -85,B 0,C 180,E1 -6906.903,E2 -6906.903} C_VEL
LIN {X 0,Y 482.934,Z 245.581,A -85,B 0,C 180,E1 -6910.002,E2 -6910.002} C_VEL
LIN {X 0,Y 482.301,Z 264.431,A -85,B 0,C 180,E1 -6913.056,E2 -6913.056} C_VEL
LIN {X 0,Y 482.261,Z 267.046,A -85,B 0,C 180,E1 -6913.447,E2 -6913.447} C_VEL
LIN {X 0,Y 484.864,Z 284.649,A -85,B 0,C 180,E1 -6913.812,E2 -6913.812} C_VEL
LIN {X 0,Y 484.263,Z 376.169,A -85,B 0,C 180,E1 -6915.207,E2 -6915.207} C_VEL
LIN {X 0,Y 483.884,Z 389.965,A -85,B 0,C 180,E1 -6915.598,E2 -6915.598} C_VEL
LIN {X 0,Y 483.409,Z 402.359,A -85,B 0,C 180,E1 -6916.12,E2 -6916.12} C_VEL
LIN {X 0,Y 482.982,Z 415.039,A -85,B 0,C 180,E1 -6916.858,E2 -6916.858} C_VEL
LIN {X 0,Y 482.488,Z 426.352,A -85,B 0,C 180,E1 -6917.702,E2 -6917.702} C_VEL
LIN {X 0,Y 482.086,Z 436.507,A -85,B 0,C 180,E1 -6918.649,E2 -6918.649} C_VEL
LIN {X 0,Y 481.692,Z 445.689,A -85,B 0,C 180,E1 -6919.704,E2 -6919.704} C_VEL
LIN {X 0,Y 481.348,Z 454.649,A -85,B 0,C 180,E1 -6920.969,E2 -6920.969} C_VEL
LIN {X 0,Y 481.095,Z 461.876,A -85,B 0,C 180,E1 -6922.233,E2 -6922.233} C_VEL
LIN {X 0,Y 481.015,Z 467.592,A -85,B 0,C 180,E1 -6923.482,E2 -6923.482} C_VEL
LIN {X 0,Y 480.894,Z 472.829,A -85,B 0,C 180,E1 -6924.968,E2 -6924.968} C_VEL
LIN {X 0,Y 480.831,Z 475.139,A -85,B 0,C 180,E1 -6925.808,E2 -6925.808} C_VEL
LIN {X 0,Y 480.889,Z 477.016,A -85,B 0,C 180,E1 -6926.648,E2 -6926.648} C_VEL
LIN {X 0,Y 480.845,Z 478.42,A -85,B 0,C 180,E1 -6927.486,E2 -6927.486} C_VEL
LIN {X 0,Y 480.823,Z 479.424,A -85,B 0,C 180,E1 -6928.324,E2 -6928.324} C_VEL
LIN {X 0,Y 480.753,Z 480.255,A -85,B 0,C 180,E1 -6929.999,E2 -6929.999} C_VEL
LIN {X 0,Y 480.823,Z 479.434,A -85,B 0,C 180,E1 -6931.674,E2 -6931.674} C_VEL
LIN {X 0,Y 480.845,Z 478.436,A -85,B 0,C 180,E1 -6932.511,E2 -6932.511} C_VEL
LIN {X 0,Y 480.888,Z 477.034,A -85,B 0,C 180,E1 -6933.35,E2 -6933.35} C_VEL
LIN {X 0,Y 480.837,Z 474.08,A -85,B 0,C 180,E1 -6934.609,E2 -6934.609} C_VEL
LIN {X 0,Y 480.914,Z 470.084,A -85,B 0,C 180,E1 -6935.869,E2 -6935.869} C_VEL
LIN {X 0,Y 481.049,Z 463.934,A -85,B 0,C 180,E1 -6937.342,E2 -6937.342} C_VEL
LIN {X 0,Y 481.286,Z 457.218,A -85,B 0,C 180,E1 -6938.606,E2 -6938.606} C_VEL
LIN {X 0,Y 481.542,Z 448.884,A -85,B 0,C 180,E1 -6939.872,E2 -6939.872} C_VEL
LIN {X 0,Y 481.909,Z 440.334,A -85,B 0,C 180,E1 -6940.926,E2 -6940.926} C_VEL
LIN {X 0,Y 482.382,Z 429.811,A -85,B 0,C 180,E1 -6941.975,E2 -6941.975} C_VEL
LIN {X 0,Y 482.824,Z 417.997,A -85,B 0,C 180,E1 -6942.919,E2 -6942.919} C_VEL
LIN {X 0,Y 483.272,Z 405.811,A -85,B 0,C 180,E1 -6943.666,E2 -6943.666} C_VEL
LIN {X 0,Y 483.679,Z 393.278,A -85,B 0,C 180,E1 -6944.244,E2 -6944.244} C_VEL
LIN {X 0,Y 484.048,Z 380.21,A -85,B 0,C 180,E1 -6944.663,E2 -6944.663} C_VEL
LIN {X 0,Y 484.289,Z 364.416,A -85,B 0,C 180,E1 -6944.951,E2 -6944.951} C_VEL
LIN {X 0,Y 484.653,Z 283.832,A -85,B 0,C 180,E1 -6946.156,E2 -6946.156} C_VEL
LIN {X 0,Y 482.215,Z 266.982,A -85,B 0,C 180,E1 -6946.508,E2 -6946.508} C_VEL
LIN {X 0,Y 482.769,Z 249.37,A -85,B 0,C 180,E1 -6949.344,E2 -6949.344} C_VEL
LIN {X 0,Y 483.436,Z 230.383,A -85,B 0,C 180,E1 -6952.43,E2 -6952.43} C_VEL
LIN {X 0,Y 483.77,Z 220.833,A -85,B 0,C 180,E1 -6953.998,E2 -6953.998} C_VEL
LIN {X 0,Y 481.727,Z 209.482,A -85,B 0,C 180,E1 -6956.01,E2 -6956.01} C_VEL
LIN {X 0,Y 481.664,Z 209.486,A -85,B 0,C 180,E1 -6958.899,E2 -6958.899} C_VEL
LIN {X 0,Y 481.641,Z 209.492,A -85,B 0,C 180,E1 -6962.185,E2 -6962.185} C_VEL
LIN {X 0,Y 481.674,Z 209.482,A -85,B 0,C 180,E1 -6964.678,E2 -6964.678} C_VEL
LIN {X 0,Y 481.633,Z 209.494,A -85,B 0,C 180,E1 -6968.003,E2 -6968.003} C_VEL
LIN {X 0,Y 481.631,Z 209.486,A -85,B 0,C 180,E1 -6971.038,E2 -6971.038} C_VEL
LIN {X 0,Y 481.631,Z 209.488,A -85,B 0,C 180,E1 -6974.454,E2 -6974.454} C_VEL
LIN {X 0,Y 481.658,Z 209.483,A -85,B 0,C 180,E1 -6976.842,E2 -6976.842} C_VEL
LIN {X 0,Y 481.68,Z 209.484,A -85,B 0,C 180,E1 -6980.06,E2 -6980.06} C_VEL
LIN {X 0,Y 481.594,Z 209.495,A -85,B 0,C 180,E1 -6983.372,E2 -6983.372} C_VEL
LIN {X 0,Y 481.671,Z 209.482,A -85,B 0,C 180,E1 -6986.327,E2 -6986.327} C_VEL
LIN {X 0,Y 481.616,Z 209.494,A -85,B 0,C 180,E1 -6989.413,E2 -6989.413} C_VEL
LIN {X 0,Y 481.659,Z 209.484,A -85,B 0,C 180,E1 -6992.165,E2 -6992.165} C_VEL
LIN {X 0,Y 481.677,Z 209.482,A -85,B 0,C 180,E1 -6994.967,E2 -6994.967} C_VEL
LIN {X 0,Y 481.628,Z 209.492,A -85,B 0,C 180,E1 -6997.703,E2 -6997.703} C_VEL
LIN {X 0,Y 481.659,Z 209.483,A -85,B 0,C 180,E1 -7000.391,E2 -7000.391} C_VEL
LIN {X 0,Y 481.647,Z 209.488,A -85,B 0,C 180,E1 -7003.032,E2 -7003.032} C_VEL
LIN {X 0,Y 481.645,Z 209.488,A -85,B 0,C 180,E1 -7005.637,E2 -7005.637} C_VEL
LIN {X 0,Y 481.745,Z 209.472,A -85,B 0,C 180,E1 -7008.215,E2 -7008.215} C_VEL
LIN {X 0,Y 481.736,Z 209.476,A -85,B 0,C 180,E1 -7011.611,E2 -7011.611} C_VEL
LIN {X 0,Y 481.782,Z 209.467,A -85,B 0,C 180,E1 -7014.139,E2 -7014.139} C_VEL
LIN {X 0,Y 481.873,Z 209.459,A -85,B 0,C 180,E1 -7017.492,E2 -7017.492} C_VEL
LIN {X 0,Y 481.881,Z 209.455,A -85,B 0,C 180,E1 -7020,E2 -7020} C_VEL
LIN {X 0,Y 481.872,Z 209.458,A -85,B 0,C 180,E1 -7022.507,E2 -7022.507} C_VEL
LIN {X 0,Y 481.757,Z 209.471,A -85,B 0,C 180,E1 -7025.861,E2 -7025.861} C_VEL
LIN {X 0,Y 481.709,Z 209.478,A -85,B 0,C 180,E1 -7028.389,E2 -7028.389} C_VEL
LIN {X 0,Y 481.743,Z 209.472,A -85,B 0,C 180,E1 -7031.785,E2 -7031.785} C_VEL
LIN {X 0,Y 481.673,Z 209.481,A -85,B 0,C 180,E1 -7035.66,E2 -7035.66} C_VEL
LIN {X 0,Y 481.661,Z 209.491,A -85,B 0,C 180,E1 -7038.723,E2 -7038.723} C_VEL
LIN {X 0,Y 481.603,Z 209.49,A -85,B 0,C 180,E1 -7041.396,E2 -7041.396} C_VEL
LIN {X 0,Y 481.632,Z 209.488,A -85,B 0,C 180,E1 -7044.115,E2 -7044.115} C_VEL
LIN {X 0,Y 481.7,Z 209.479,A -85,B 0,C 180,E1 -7047.142,E2 -7047.142} C_VEL
LIN {X 0,Y 481.633,Z 209.486,A -85,B 0,C 180,E1 -7049.744,E2 -7049.744} C_VEL
LIN {X 0,Y 481.629,Z 209.493,A -85,B 0,C 180,E1 -7052.677,E2 -7052.677} C_VEL
LIN {X 0,Y 481.602,Z 209.49,A -85,B 0,C 180,E1 -7055.712,E2 -7055.712} C_VEL
LIN {X 0,Y 481.632,Z 209.489,A -85,B 0,C 180,E1 -7058.863,E2 -7058.863} C_VEL
LIN {X 0,Y 481.618,Z 209.491,A -85,B 0,C 180,E1 -7061.916,E2 -7061.916} C_VEL
LIN {X 0,Y 481.622,Z 209.494,A -85,B 0,C 180,E1 -7064.461,E2 -7064.461} C_VEL
LIN {X 0,Y 481.618,Z 209.491,A -85,B 0,C 180,E1 -7067.843,E2 -7067.843} C_VEL
LIN {X 0,Y 481.652,Z 209.486,A -85,B 0,C 180,E1 -7070.655,E2 -7070.655} C_VEL
LIN {X 0,Y 481.606,Z 209.49,A -85,B 0,C 180,E1 -7073.379,E2 -7073.379} C_VEL
LIN {X 0,Y 481.688,Z 209.484,A -85,B 0,C 180,E1 -7076.334,E2 -7076.334} C_VEL
LIN {X 0,Y 481.631,Z 209.487,A -85,B 0,C 180,E1 -7079.421,E2 -7079.421} C_VEL
LIN {X 0,Y 481.682,Z 209.486,A -85,B 0,C 180,E1 -7082.171,E2 -7082.171} C_VEL
LIN {X 0,Y 481.678,Z 209.48,A -85,B 0,C 180,E1 -7084.972,E2 -7084.972} C_VEL
LIN {X 0,Y 481.621,Z 209.49,A -85,B 0,C 180,E1 -7088.016,E2 -7088.016} C_VEL
LIN {X 0,Y 480.957,Z 209.572,A -85,B 0,C 180,E1 -7088.714,E2 -7088.714} C_VEL
LIN {X 0,Y 478.131,Z 209.93,A -85,B 0,C 180,E1 -7089.848,E2 -7089.848} C_VEL
LIN {X 0,Y 475.743,Z 210.223,A -85,B 0,C 180,E1 -7090.762,E2 -7090.762} C_VEL
LIN {X 0,Y 474.718,Z 210.351,A -85,B 0,C 180,E1 -7091.468,E2 -7091.468} C_VEL
LIN {X 0,Y 474.634,Z 210.363,A -85,B 0,C 180,E1 -7091.707,E2 -7091.707} C_VEL
LIN {X 0,Y 474.69,Z 210.351,A -85,B 0,C 180,E1 -7094.547,E2 -7094.547} C_VEL
LIN {X 0,Y 474.699,Z 210.354,A -85,B 0,C 180,E1 -7098.04,E2 -7098.04} C_VEL
LIN {X 0,Y 474.708,Z 210.354,A -85,B 0,C 180,E1 -7101.488,E2 -7101.488} C_VEL
LIN {X 0,Y 474.743,Z 210.35,A -85,B 0,C 180,E1 -7104.906,E2 -7104.906} C_VEL
LIN {X 0,Y 474.727,Z 210.39,A -85,B 0,C 180,E1 -7105.225,E2 -7105.225} C_VEL
LIN {X 0,Y 475.503,Z 217.063,A -85,B 0,C 180,E1 -7106.612,E2 -7106.612} C_VEL
LIN {X 0,Y 475.408,Z 225.716,A -85,B 0,C 180,E1 -7108.349,E2 -7108.349} C_VEL
LIN {X 0,Y 478.131,Z 240.289,A -85,B 0,C 180,E1 -7108.673,E2 -7108.673} C_VEL
LIN {X 0,Y 477.401,Z 332.432,A -85,B 0,C 180,E1 -7110.081,E2 -7110.081} C_VEL
LIN {X 0,Y 477.17,Z 344.892,A -85,B 0,C 180,E1 -7110.423,E2 -7110.423} C_VEL
LIN {X 0,Y 476.849,Z 357.73,A -85,B 0,C 180,E1 -7110.951,E2 -7110.951} C_VEL
LIN {X 0,Y 476.524,Z 369.116,A -85,B 0,C 180,E1 -7111.586,E2 -7111.586} C_VEL
LIN {X 0,Y 475.975,Z 380.873,A -85,B 0,C 180,E1 -7112.434,E2 -7112.434} C_VEL
LIN {X 0,Y 475.529,Z 391.359,A -85,B 0,C 180,E1 -7113.39,E2 -7113.39} C_VEL
LIN {X 0,Y 475.098,Z 400.835,A -85,B 0,C 180,E1 -7114.455,E2 -7114.455} C_VEL
LIN {X 0,Y 474.703,Z 409.959,A -85,B 0,C 180,E1 -7115.736,E2 -7115.736} C_VEL
LIN {X 0,Y 474.429,Z 417.301,A -85,B 0,C 180,E1 -7117.019,E2 -7117.019} C_VEL
LIN {X 0,Y 474.12,Z 424.095,A -85,B 0,C 180,E1 -7118.525,E2 -7118.525} C_VEL
LIN {X 0,Y 473.963,Z 428.569,A -85,B 0,C 180,E1 -7119.819,E2 -7119.819} C_VEL
LIN {X 0,Y 473.843,Z 431.965,A -85,B 0,C 180,E1 -7121.118,E2 -7121.118} C_VEL
LIN {X 0,Y 473.793,Z 433.651,A -85,B 0,C 180,E1 -7121.986,E2 -7121.986} C_VEL
LIN {X 0,Y 473.711,Z 434.934,A -85,B 0,C 180,E1 -7122.859,E2 -7122.859} C_VEL
LIN {X 0,Y 473.676,Z 435.797,A -85,B 0,C 180,E1 -7123.733,E2 -7123.733} C_VEL
LIN {X 0,Y 473.707,Z 436.243,A -85,B 0,C 180,E1 -7125.346,E2 -7125.346} C_VEL
LIN {X 0,Y 473.655,Z 435.83,A -85,B 0,C 180,E1 -7126.375,E2 -7126.375} C_VEL
LIN {X 0,Y 473.695,Z 434.978,A -85,B 0,C 180,E1 -7127.261,E2 -7127.261} C_VEL
LIN {X 0,Y 473.804,Z 433.398,A -85,B 0,C 180,E1 -7128.32,E2 -7128.32} C_VEL
LIN {X 0,Y 473.929,Z 429.721,A -85,B 0,C 180,E1 -7129.942,E2 -7129.942} C_VEL
LIN {X 0,Y 474.103,Z 425.378,A -85,B 0,C 180,E1 -7131.295,E2 -7131.295} C_VEL
LIN {X 0,Y 474.337,Z 419.697,A -85,B 0,C 180,E1 -7132.657,E2 -7132.657} C_VEL
LIN {X 0,Y 474.677,Z 412.476,A -85,B 0,C 180,E1 -7134.026,E2 -7134.026} C_VEL
LIN {X 0,Y 475.027,Z 404.957,A -85,B 0,C 180,E1 -7135.172,E2 -7135.172} C_VEL
LIN {X 0,Y 475.471,Z 395.667,A -85,B 0,C 180,E1 -7136.322,E2 -7136.322} C_VEL
LIN {X 0,Y 475.934,Z 385.218,A -85,B 0,C 180,E1 -7137.37,E2 -7137.37} C_VEL
LIN {X 0,Y 476.399,Z 375.348,A -85,B 0,C 180,E1 -7138.168,E2 -7138.168} C_VEL
LIN {X 0,Y 476.86,Z 363.626,A -85,B 0,C 180,E1 -7138.919,E2 -7138.919} C_VEL
LIN {X 0,Y 477.199,Z 351.899,A -85,B 0,C 180,E1 -7139.491,E2 -7139.491} C_VEL
LIN {X 0,Y 477.468,Z 338.781,A -85,B 0,C 180,E1 -7139.946,E2 -7139.946} C_VEL
LIN {X 0,Y 477.595,Z 324.806,A -85,B 0,C 180,E1 -7140.233,E2 -7140.233} C_VEL
LIN {X 0,Y 478.267,Z 239.147,A -85,B 0,C 180,E1 -7141.538,E2 -7141.538} C_VEL
LIN {X 0,Y 475.556,Z 225.786,A -85,B 0,C 180,E1 -7141.87,E2 -7141.87} C_VEL
LIN {X 0,Y 475.647,Z 215.62,A -85,B 0,C 180,E1 -7143.884,E2 -7143.884} C_VEL
LIN {X 0,Y 474.67,Z 210.359,A -85,B 0,C 180,E1 -7145.009,E2 -7145.009} C_VEL
LIN {X 0,Y 474.612,Z 210.369,A -85,B 0,C 180,E1 -7148.455,E2 -7148.455} C_VEL
LIN {X 0,Y 474.635,Z 210.359,A -85,B 0,C 180,E1 -7150.961,E2 -7150.961} C_VEL
LIN {X 0,Y 474.604,Z 210.369,A -85,B 0,C 180,E1 -7154.102,E2 -7154.102} C_VEL
LIN {X 0,Y 474.636,Z 210.36,A -85,B 0,C 180,E1 -7157.069,E2 -7157.069} C_VEL
LIN {X 0,Y 474.65,Z 210.361,A -85,B 0,C 180,E1 -7160.455,E2 -7160.455} C_VEL
LIN {X 0,Y 474.572,Z 210.369,A -85,B 0,C 180,E1 -7163.675,E2 -7163.675} C_VEL
LIN {X 0,Y 474.622,Z 210.36,A -85,B 0,C 180,E1 -7166.779,E2 -7166.779} C_VEL
LIN {X 0,Y 474.59,Z 210.369,A -85,B 0,C 180,E1 -7169.769,E2 -7169.769} C_VEL
LIN {X 0,Y 474.673,Z 210.353,A -85,B 0,C 180,E1 -7172.679,E2 -7172.679} C_VEL
LIN {X 0,Y 474.641,Z 210.358,A -85,B 0,C 180,E1 -7175.506,E2 -7175.506} C_VEL
LIN {X 0,Y 474.649,Z 210.354,A -85,B 0,C 180,E1 -7179.185,E2 -7179.185} C_VEL
LIN {X 0,Y 474.63,Z 210.361,A -85,B 0,C 180,E1 -7181.884,E2 -7181.884} C_VEL
LIN {X 0,Y 474.671,Z 210.354,A -85,B 0,C 180,E1 -7184.544,E2 -7184.544} C_VEL
LIN {X 0,Y 474.675,Z 210.354,A -85,B 0,C 180,E1 -7188.037,E2 -7188.037} C_VEL
LIN {X 0,Y 474.699,Z 210.352,A -85,B 0,C 180,E1 -7191.486,E2 -7191.486} C_VEL
LIN {X 0,Y 474.76,Z 210.343,A -85,B 0,C 180,E1 -7194.052,E2 -7194.052} C_VEL
LIN {X 0,Y 474.861,Z 210.334,A -85,B 0,C 180,E1 -7197.455,E2 -7197.455} C_VEL
LIN {X 0,Y 474.825,Z 210.334,A -85,B 0,C 180,E1 -7200.848,E2 -7200.848} C_VEL
LIN {X 0,Y 474.86,Z 210.327,A -85,B 0,C 180,E1 -7202.545,E2 -7202.545} C_VEL
LIN {X 0,Y 474.734,Z 210.34,A -85,B 0,C 180,E1 -7205.948,E2 -7205.948} C_VEL
LIN {X 0,Y 474.681,Z 210.352,A -85,B 0,C 180,E1 -7208.515,E2 -7208.515} C_VEL
LIN {X 0,Y 474.71,Z 210.347,A -85,B 0,C 180,E1 -7211.963,E2 -7211.963} C_VEL
LIN {X 0,Y 474.651,Z 210.354,A -85,B 0,C 180,E1 -7215.768,E2 -7215.768} C_VEL
LIN {X 0,Y 474.634,Z 210.36,A -85,B 0,C 180,E1 -7219.012,E2 -7219.012} C_VEL
LIN {X 0,Y 474.56,Z 210.367,A -85,B 0,C 180,E1 -7221.731,E2 -7221.731} C_VEL
LIN {X 0,Y 474.6,Z 210.365,A -85,B 0,C 180,E1 -7224.496,E2 -7224.496} C_VEL
LIN {X 0,Y 474.614,Z 210.359,A -85,B 0,C 180,E1 -7227.326,E2 -7227.326} C_VEL
LIN {X 0,Y 474.578,Z 210.369,A -85,B 0,C 180,E1 -7230.232,E2 -7230.232} C_VEL
LIN {X 0,Y 474.594,Z 210.364,A -85,B 0,C 180,E1 -7233.224,E2 -7233.224} C_VEL
LIN {X 0,Y 474.564,Z 210.374,A -85,B 0,C 180,E1 -7236.326,E2 -7236.326} C_VEL
LIN {X 0,Y 474.606,Z 210.363,A -85,B 0,C 180,E1 -7239.55,E2 -7239.55} C_VEL
LIN {X 0,Y 474.588,Z 210.362,A -85,B 0,C 180,E1 -7242.235,E2 -7242.235} C_VEL
LIN {X 0,Y 474.604,Z 210.362,A -85,B 0,C 180,E1 -7245.3,E2 -7245.3} C_VEL
LIN {X 0,Y 474.598,Z 210.37,A -85,B 0,C 180,E1 -7248.215,E2 -7248.215} C_VEL
LIN {X 0,Y 474.601,Z 210.365,A -85,B 0,C 180,E1 -7251.544,E2 -7251.544} C_VEL
LIN {X 0,Y 474.619,Z 210.363,A -85,B 0,C 180,E1 -7254.727,E2 -7254.727} C_VEL
LIN {X 0,Y 474.631,Z 210.364,A -85,B 0,C 180,E1 -7257.789,E2 -7257.789} C_VEL
LIN {X 0,Y 474.604,Z 210.365,A -85,B 0,C 180,E1 -7260.89,E2 -7260.89} C_VEL
LIN {X 0,Y 474.656,Z 210.477,A -85,B 0,C 180,E1 -7263.658,E2 -7263.658} C_VEL
LIN {X 0,Y 476.785,Z 221.139,A -85,B 0,C 180,E1 -7265.624,E2 -7265.624} C_VEL
LIN {X 0,Y 476.833,Z 226.532,A -85,B 0,C 180,E1 -7266.551,E2 -7266.551} C_VEL
LIN {X 0,Y 476.054,Z 244.019,A -85,B 0,C 180,E1 -7269.475,E2 -7269.475} C_VEL
LIN {X 0,Y 475.43,Z 261.516,A -85,B 0,C 180,E1 -7272.36,E2 -7272.36} C_VEL
LIN {X 0,Y 475.256,Z 266.479,A -85,B 0,C 180,E1 -7273.172,E2 -7273.172} C_VEL
LIN {X 0,Y 478.1,Z 286.038,A -85,B 0,C 180,E1 -7273.586,E2 -7273.586} C_VEL
LIN {X 0,Y 477.432,Z 375.228,A -85,B 0,C 180,E1 -7274.963,E2 -7274.963} C_VEL
LIN {X 0,Y 477.066,Z 388.454,A -85,B 0,C 180,E1 -7275.333,E2 -7275.333} C_VEL
LIN {X 0,Y 476.583,Z 401.175,A -85,B 0,C 180,E1 -7275.863,E2 -7275.863} C_VEL
LIN {X 0,Y 476.107,Z 413.297,A -85,B 0,C 180,E1 -7276.556,E2 -7276.556} C_VEL
LIN {X 0,Y 475.655,Z 424.272,A -85,B 0,C 180,E1 -7277.364,E2 -7277.364} C_VEL
LIN {X 0,Y 475.169,Z 435.253,A -85,B 0,C 180,E1 -7278.374,E2 -7278.374} C_VEL
LIN {X 0,Y 474.735,Z 443.777,A -85,B 0,C 180,E1 -7279.335,E2 -7279.335} C_VEL
LIN {X 0,Y 474.342,Z 453.028,A -85,B 0,C 180,E1 -7280.62,E2 -7280.62} C_VEL
LIN {X 0,Y 474.085,Z 460.478,A -85,B 0,C 180,E1 -7281.903,E2 -7281.903} C_VEL
LIN {X 0,Y 473.902,Z 466.467,A -85,B 0,C 180,E1 -7283.185,E2 -7283.185} C_VEL
LIN {X 0,Y 473.834,Z 471.205,A -85,B 0,C 180,E1 -7284.467,E2 -7284.467} C_VEL
LIN {X 0,Y 473.737,Z 474.825,A -85,B 0,C 180,E1 -7285.745,E2 -7285.745} C_VEL
LIN {X 0,Y 473.796,Z 476.698,A -85,B 0,C 180,E1 -7286.597,E2 -7286.597} C_VEL
LIN {X 0,Y 473.756,Z 479.102,A -85,B 0,C 180,E1 -7288.299,E2 -7288.299} C_VEL
LIN {X 0,Y 473.679,Z 479.929,A -85,B 0,C 180,E1 -7289.999,E2 -7289.999} C_VEL
LIN {X 0,Y 473.756,Z 479.104,A -85,B 0,C 180,E1 -7291.699,E2 -7291.699} C_VEL
LIN {X 0,Y 473.761,Z 478.104,A -85,B 0,C 180,E1 -7292.549,E2 -7292.549} C_VEL
LIN {X 0,Y 473.795,Z 476.697,A -85,B 0,C 180,E1 -7293.4,E2 -7293.4} C_VEL
LIN {X 0,Y 473.76,Z 473.738,A -85,B 0,C 180,E1 -7294.678,E2 -7294.678} C_VEL
LIN {X 0,Y 473.822,Z 469.732,A -85,B 0,C 180,E1 -7295.958,E2 -7295.958} C_VEL
LIN {X 0,Y 473.983,Z 463.564,A -85,B 0,C 180,E1 -7297.452,E2 -7297.452} C_VEL
LIN {X 0,Y 474.197,Z 456.828,A -85,B 0,C 180,E1 -7298.736,E2 -7298.736} C_VEL
LIN {X 0,Y 474.483,Z 448.469,A -85,B 0,C 180,E1 -7300.02,E2 -7300.02} C_VEL
LIN {X 0,Y 474.905,Z 439.883,A -85,B 0,C 180,E1 -7301.089,E2 -7301.089} C_VEL
LIN {X 0,Y 475.371,Z 429.568,A -85,B 0,C 180,E1 -7302.133,E2 -7302.133} C_VEL
LIN {X 0,Y 475.803,Z 418.773,A -85,B 0,C 180,E1 -7303.015,E2 -7303.015} C_VEL
LIN {X 0,Y 476.256,Z 407.211,A -85,B 0,C 180,E1 -7303.763,E2 -7303.763} C_VEL
LIN {X 0,Y 476.694,Z 395.22,A -85,B 0,C 180,E1 -7304.349,E2 -7304.349} C_VEL
LIN {X 0,Y 477.095,Z 382.264,A -85,B 0,C 180,E1 -7304.8,E2 -7304.8} C_VEL
LIN {X 0,Y 477.388,Z 370.182,A -85,B 0,C 180,E1 -7305.063,E2 -7305.063} C_VEL
LIN {X 0,Y 477.833,Z 284.834,A -85,B 0,C 180,E1 -7306.358,E2 -7306.358} C_VEL
LIN {X 0,Y 475.237,Z 266.774,A -85,B 0,C 180,E1 -7306.723,E2 -7306.723} C_VEL
LIN {X 0,Y 475.799,Z 249.099,A -85,B 0,C 180,E1 -7309.61,E2 -7309.61} C_VEL
LIN {X 0,Y 476.468,Z 231.291,A -85,B 0,C 180,E1 -7312.547,E2 -7312.547} C_VEL
LIN {X 0,Y 476.812,Z 221.955,A -85,B 0,C 180,E1 -7314.102,E2 -7314.102} C_VEL
LIN {X 0,Y 474.72,Z 210.355,A -85,B 0,C 180,E1 -7316.2,E2 -7316.2} C_VEL
LIN {X 0,Y 474.607,Z 210.366,A -85,B 0,C 180,E1 -7319.248,E2 -7319.248} C_VEL
LIN {X 0,Y 474.599,Z 210.366,A -85,B 0,C 180,E1 -7322.427,E2 -7322.427} C_VEL
LIN {X 0,Y 474.6,Z 210.364,A -85,B 0,C 180,E1 -7325.466,E2 -7325.466} C_VEL
LIN {X 0,Y 474.589,Z 210.366,A -85,B 0,C 180,E1 -7328.453,E2 -7328.453} C_VEL
LIN {X 0,Y 474.603,Z 210.362,A -85,B 0,C 180,E1 -7330.955,E2 -7330.955} C_VEL
LIN {X 0,Y 474.581,Z 210.369,A -85,B 0,C 180,E1 -7334.101,E2 -7334.101} C_VEL
LIN {X 0,Y 474.621,Z 210.36,A -85,B 0,C 180,E1 -7337.066,E2 -7337.066} C_VEL
LIN {X 0,Y 474.649,Z 210.357,A -85,B 0,C 180,E1 -7340.454,E2 -7340.454} C_VEL
LIN {X 0,Y 474.556,Z 210.376,A -85,B 0,C 180,E1 -7343.673,E2 -7343.673} C_VEL
LIN {X 0,Y 474.604,Z 210.362,A -85,B 0,C 180,E1 -7346.777,E2 -7346.777} C_VEL
LIN {X 0,Y 474.572,Z 210.371,A -85,B 0,C 180,E1 -7349.767,E2 -7349.767} C_VEL
LIN {X 0,Y 474.654,Z 210.355,A -85,B 0,C 180,E1 -7352.677,E2 -7352.677} C_VEL
LIN {X 0,Y 474.622,Z 210.368,A -85,B 0,C 180,E1 -7355.505,E2 -7355.505} C_VEL
LIN {X 0,Y 474.628,Z 210.363,A -85,B 0,C 180,E1 -7359.183,E2 -7359.183} C_VEL
LIN {X 0,Y 474.609,Z 210.363,A -85,B 0,C 180,E1 -7361.882,E2 -7361.882} C_VEL
LIN {X 0,Y 474.649,Z 210.356,A -85,B 0,C 180,E1 -7364.542,E2 -7364.542} C_VEL
LIN {X 0,Y 474.688,Z 210.352,A -85,B 0,C 180,E1 -7368.037,E2 -7368.037} C_VEL
LIN {X 0,Y 474.695,Z 210.355,A -85,B 0,C 180,E1 -7371.486,E2 -7371.486} C_VEL
LIN {X 0,Y 474.744,Z 210.344,A -85,B 0,C 180,E1 -7374.052,E2 -7374.052} C_VEL
LIN {X 0,Y 474.84,Z 210.336,A -85,B 0,C 180,E1 -7377.455,E2 -7377.455} C_VEL
LIN {X 0,Y 474.822,Z 210.34,A -85,B 0,C 180,E1 -7380.848,E2 -7380.848} C_VEL
LIN {X 0,Y 474.838,Z 210.335,A -85,B 0,C 180,E1 -7382.545,E2 -7382.545} C_VEL
LIN {X 0,Y 474.719,Z 210.347,A -85,B 0,C 180,E1 -7385.948,E2 -7385.948} C_VEL
LIN {X 0,Y 474.674,Z 210.356,A -85,B 0,C 180,E1 -7388.514,E2 -7388.514} C_VEL
